bQARowStopperMotorFwd1:=FALSE;
bQARowStopperMotorFwd2:=FALSE;
bQARowStopperMotorFwd3:=FALSE;
bQARowStopperMotorRev1:=FALSE;
bQARowStopperMotorRev2:=FALSE;
bQARowStopperMotorRev3:=FALSE;
bQARowStopperMotorRevAuto:=FALSE;
bRowStopperGoRst:=FALSE;
step2:=0;
step1:=0;
step3:=0;
step4:=0;

END_IF
END_PROGRAM

(* POU Auto/ColumStopperMotor, ST *)
PROGRAM ColumStopperMotor
VAR
	bQAColumnStopperMotorFwd1: BOOL;
	bQAColumnStopperMotorRev1: BOOL;
	step1: INT;

	test: BOOL;

	step2: INT;
	ColumnStopperInHome: BOOL;
	bA4_4MoveStarted: BOOL;
	bQAColumnStopperMotorFw21: BOOL;
	bQAColumnStopperMotorFwd2: BOOL;
	bQAColumnStopperMotorRev2: BOOL;
	bQAColumnStopperMotorFw2: BOOL;
	test1: BOOL;
	step3: INT;
	test2: BOOL;
	bA2_3MoveStarted: BOOL;
	bQAColumnStopperMotorRev3: BOOL;
	bQAColumnStopperMotorFwd3: BOOL;
	RevOffDly: TON;
	bA2_4MoveStarted: BOOL;
	Timer1: TON;
	Timer2: TON;
	bStopHmitemp: BOOL;
	bProgramChange: BOOL;
	bColumnStopMove2_3: BOOL;
	bColumnStopMove2_4: BOOL;
	b2_3SetHmiSelectedtemp: BOOL;
	b2_4SetHmiSelectedtemp: BOOL;
	b2_4SetHmiSelectedtemp1: BOOL;
	Mybit1: BOOL;
END_VAR
bQAColumnStopperMotorForward:= ( bQAColumnStopperMotorFwd1 OR bQAColumnStopperMotorFwd2 OR bQAColumnStopperMotorFwd3  ) ;
bQAColumnStopperMotorReverse:= ( bQAColumnStopperMotorRev1 ) ;

								(*=========== Column Stopper Motor Home Position Logic===============*)

CASE step2 OF

	0:	IF  bInitializeHmi AND NOT bIColumnStopperHome  AND NOT bAinterlockinit   THEN
		bQAColumnStopperMotorFwd1:=TRUE;
		(*	Timer1(IN:=TRUE  , PT:=t#1s , Q=> , ET=> );   *) step2:=step2+1;
		ELSIF  bInitializeHmi AND  bIColumnStopperHome    THEN   step2:=4;
		END_IF

	1:	bQAColumnStopperMotorFwd1:=FALSE;
		Timer2(IN:=TRUE , PT:= t#0.5s, Q=> , ET=> );
		IF Timer2.Q THEN step2 :=step2+1; END_IF

	2:	IF NOT bAPauseSeq  THEN  bQAColumnStopperMotorRev1:=TRUE; step2:=step2+1; END_IF

	3:	IF bIColumnStopperHome THEN bQAColumnStopperMotorRev1:=FALSE; step2:=step2+1; END_IF

	4:	IF b2_3SetHmiSelected THEN bColumnStopMove2_3:=TRUE; step2:=0;
		ELSIF b2_4SetHmiSelected THEN bColumnStopMove2_4:=TRUE; step2:=0;
		END_IF

END_CASE

										(*=========== Column Stopper Motor 2_3 Position Logic===============*)

CASE step1 OF

	0:	IF  b2_3SetHmiSelected AND bColumnStopMove2_3 AND NOT bIColumnStopper3  AND  bIColumnStopperHome  THEN
		 bQAColumnStopperMotorFwd2:=TRUE; step1:=step1+1;
		END_IF

	1:	IF bIColumnStopper3 THEN
	         bColumnStopMove2_3:=FALSE;
                  bQAColumnStopperMotorFwd2:=FALSE; step1:=step1+1;
		END_IF

	2:	 step1:=0;

END_CASE

										(*=========== Column Stopper Motor 2_4 Position Logic===============*)

CASE step3 OF

	0:	IF b2_4SetHmiSelected AND  bColumnStopMove2_4 AND NOT bIColumnStopper2  AND    bIColumnStopperHome   THEN
		bQAColumnStopperMotorFwd3:=TRUE; step3:=step3+1;
		END_IF


	1: 	IF bIColumnStopper2 THEN
		bColumnStopMove2_4:=FALSE;
		bQAColumnStopperMotorFwd3:=FALSE; step3:=step3+1;
		END_IF


	2:	step3:=0;

END_CASE
END_PROGRAM

(* POU StartUp/GripperUnitRst, ST *)
PROGRAM GripperUnitRst
VAR
	step: INT;
	bILengthTightPistonEnd: BOOL;
	bIBredthTightPistonEnd: BOOL;
	bEmptyCortonConveyoPiatonHome: BOOL;
	bHorPistonAtReadyPos: BOOL;
	bHorPistonAtHomePos: BOOL;
	bHorPistonAtMiddlePos: BOOL;
	bGripperAtHomePos: BOOL;
	bGripperAtEndPos: BOOL;
	bGripperAtMiddlePos: BOOL;
	bSepVerticalAtHomePos: BOOL;
	bSepVerticalAtEndPos: BOOL;
	bSepVerticalAtMiddlePos: BOOL;
	bLenghtTightPistonHomeNok: BOOL;
	bBreathtightPistonHomeNok: BOOL;
	bApplicatorHomeNok: BOOL;
	bReleaseApplicator: BOOL;
	step2: INT;
	Timer1: TON;
	Timer2: TON;
	Timer3: TON;
	Timer4: TON;
	ReadyToRelease: BOOL;
	Timer5: TON;
	bAResetHmitemp: BOOL;
	Timer6: TON;
	Timer7: TON;
	Timer8: TON;
	Timer9: TON;
	test: BOOL;
END_VAR
VAR_INPUT
END_VAR
IF bInitializeHmi AND bAutoModeOn AND bMCStartInAuto THEN
step:=0;
END_IF



CASE step OF
	0:	iControlWord1.7:=TRUE;
		 bHomingDone:=FALSE;
		step:=step+1;

	1:	 iControlWord1.7:=FALSE;
		step:=step+1;


	2:	IF  bAResetHmitemp OR bMatrixConvIntOver THEN step:=step+1;  END_IF

	3:	IF NOT bIGripperVerticalHome THEN   bRServoHome:=TRUE; step:=step+1;
		ELSIF bIGripperVerticalHome  THEN step:=5;
		END_IF

	4:	IF bHomingDone THEN step:=step+1; END_IF

	5:	bMatrixConvIntOver:=FALSE;
		bHomingDone:=FALSE; (*bRowStopperGoHome:=TRUE;*)
		step:=step+1;

	6:	IF bISeparatorHorizontalPistonEnd AND NOT  bISeparatorHorizontalPistonHome THEN
		bHorPistonAtReadyPos:=TRUE; bHorPistonAtHomePos:=FALSE; bHorPistonAtMiddlePos:=FALSE;
		step:=step+1;
		ELSIF NOT bISeparatorHorizontalPistonEnd  AND  bISeparatorHorizontalPistonHome THEN
		bHorPistonAtHomePos:=TRUE; bHorPistonAtReadyPos:=FALSE; bHorPistonAtMiddlePos:=FALSE;
		step:=step+1;
		ELSIF NOT bISeparatorHorizontalPistonEnd  AND  NOT bISeparatorHorizontalPistonHome THEN
		bHorPistonAtMiddlePos:=TRUE; bHorPistonAtHomePos:=FALSE; bHorPistonAtReadyPos:=FALSE;
		step:=step+1;
		END_IF

	7:	IF bHorPistonAtReadyPos THEN step:=8;
		ELSIF bHorPistonAtHomePos THEN step:=25;
		ELSIF bHorPistonAtMiddlePos THEN  step:=25; END_IF

	8:	 iControlWord1:=0;
		step:=step+1;

	9:	 iControlWord1:=6;
		step:=Step+1;
(*========Waiting for row stopper to home==========*)

	10:	IF bIRowStopperHome THEN step:=Step+1;
		ELSIF NOT bIRowStopperHome THEN bRowStopperGoHome:=TRUE;  step:=Step+1;  END_IF


	11:	IF  bIRowStopperHome THEN iControlWord1:=7;
		bHomingDone:=FALSE;
		step:=Step+1;
		END_IF

	12:	IF ModeACT=1THEN  step:=15;
		ELSIF  ModeACT<>1 THEN step:=Step+1;
		END_IF

	13:	ModeWrite:=1;
		step:=Step+1;

	14:	bAModeWrite:=TRUE;
		Timer1(IN:=TRUE , PT:=T#100ms , Q=> , ET=> );
		IF Timer1.Q THEN step:=Step+1;  END_IF


	15:	diTargetVelocity1:=rPickVeloFinal;
		diTargetPosition:=-87947 ; (*rTargetPosFinal*);
		bAModeWrite:=FALSE;
		step:=Step+1;

	16:	Timer2(IN:=TRUE , PT:= t#100ms, Q=> , ET=> );
		IF Timer2.Q THEN  step:=Step+1; END_IF

	17:	iControlWord1:=15;
		step:=Step+1;

	18:	Timer3(IN:=TRUE , PT:= t#1s, Q=> , ET=> );
		IF Timer3.Q  THEN step:=Step+1; END_IF

	19:	IF statusWord.2 THEN    iControlWord1.4:=TRUE;
		step:=Step+1;
		END_IF
	20:	Timer4(IN:=TRUE , PT:= t#5s, Q=> , ET=> );
		IF Timer4.Q THEN iControlWord1.4:=FALSE; step:=Step+1; END_IF

	21:	IF statusWord.10 THEN step:=Step+1; END_IF

	22:	bQABreadthTightPistonValve:=FALSE;
		bQALengthTightPistonValve:=FALSE;
		bQMBreadthTightPistonValve:=FALSE;
		bQMLengthTightPistonValve:=FALSE;
		 step:=Step+1;

	23:	IF(* bILengthTightPistonHome AND*) bIBreadthTightPistonHome AND bIGripperVerticalEnd   THEN  step:=Step+1; END_IF

	24:	bRServoHome:=TRUE;
		IF bHomingDone THEN bGripperUnitOver:=TRUE;  step:=0; END_IF

(*========Reseting all auto and manual output and enabling Rst outpus===================*)

	25:	IF bIGripperVerticalHome THEN bQASeparatorHorizontalPistonValveFWD:=FALSE;
		bQASeparatorHorizontalPistonValveREV:=FALSE;
		bQMSeparatorHorizontalPistonValveRev:=FALSE;
		bQMSeparatorHorizontalPistonValveFwd:=FALSE;
		bHomingDone:=FALSE;
		step:=step+1;
		END_IF

	26:	bQRSeparatorHorizontalPistonValveREV:=TRUE;
		step:=step+1;

	27:	IF bISeparatorHorizontalPistonEnd THEN bReleaseApplicator:=TRUE; bQRSeparatorHorizontalPistonValveREV:=FALSE; step:=step+1; END_IF


	28:	IF ReadyToRelease THEN	step:=step+1; 	END_IF

	29:	Timer5(IN:=TRUE , PT:=t#1s , Q=> , ET=> );
		IF Timer5.Q THEN ReadyToRelease:=FALSE; step:=step+1; 	END_IF

	30:	bQMBreadthTightPistonValve:=FALSE;
		bQMLengthTightPistonValve:=FALSE;
		bQABreadthTightPistonValve:=FALSE;
		bQALengthTightPistonValve:=FALSE;
		step:=step+1;

	31:	IF bIBreadthTightPistonHome(* AND bILengthTightPistonHome*) THEN
		bRServoHome1:=TRUE;
		IF bHomingDone THEN bGripperUnitOver:=TRUE;  step:=0; END_IF
		END_IF


END_CASE




CASE step2 OF

	0:	IF bReleaseApplicator  THEN
		Timer6(IN:=FALSE);
		Timer7(IN:=FALSE);
		step2:=step2+1;
		END_IF

	1:	IF bIRowStopperHome THEN step2:=step2+1;
		ELSIF NOT bIRowStopperHome THEN  bRowStopperGoHome1:=TRUE;  step:=Step+1;  END_IF


	2: 	IF bIRowStopperHome  THEN   iControlWord1:=7;
		bReleaseApplicator:=FALSE;
		Timer8(IN:=FALSE);
		step2:=step2+1;
		END_IF

	3:	Timer6(IN:=TRUE , PT:=T#100ms , Q=> , ET=> );
		IF Timer6.Q THEN
		step2:=step2+1;
		END_IF

	4:	IF NOT bIGripperVerticalEnd AND bIRowStopperHome THEN
		ModeWrite:=3;							(*=========Changing the servo Mode to Velocity mode=============*)
		Timer8(IN:=FALSE);
		Timer9(IN:=FALSE);

		step2:=step2+1;
		END_IF

	5:	Timer7(IN:=TRUE , PT:=T#100ms , Q=> , ET=> );
		IF Timer7.Q THEN
		step2:=step2+1;
		END_IF


	6:	bAModeWrite:=TRUE;
		Timer8(IN:=TRUE , PT:=T#100ms , Q=> , ET=> );
		IF Timer8.Q THEN
		step2:=step2+1;
		END_IF

	7:	IF ModeWrite = ModeAct THEN
		bAModeWrite:=FALSE;
		step2:=step2+1;
		END_IF

	8:	IF  statusWord.1 THEN iControlWord1 :=15;
		Timer9(IN:=TRUE , PT:=T#1s , Q=> , ET=> );
		IF Timer9.Q THEN
		step2:=step2+1;
		END_IF
		END_IF

	9:	diTargetVelocity:=-100;
		step2:=step2+1;


	10:	IF statusWord.2 THEN
		iControlWord1.4:= TRUE;
		step2:=step2+1;
		END_IF




	11:	IF bIGripperVerticalEnd THEN
		iControlWord1.4 := FALSE;
		iControlWord1:=7;
		diTargetVelocity:=0;
		step2:=step2+1;
		END_IF

	12: 	Timer6(IN:=FALSE);
		Timer7(IN:=FALSE);
		Timer8(IN:=FALSE);
		Timer9(IN:=FALSE);
		step2:=step2+1;

	13:	ReadyToRelease:=TRUE;
		step2:=0;




END_CASE


IF NOT bIEmergencySwitch OR bStopHmi OR bIMcStop OR bServoOff  THEN

bRServoHome:=FALSE;
bHorPistonAtReadyPos:=FALSE;
bHorPistonAtHomePos:=FALSE;
bHorPistonAtMiddlePos:=FALSE;
bAModeWrite:=FALSE;
Timer1(IN:=FALSE);
Timer2(IN:=FALSE);
Timer3(IN:=FALSE);
Timer4(IN:=FALSE);
bRServoHome:=FALSE;
bQRSeparatorHorizontalPistonValveREV:=FALSE;
Timer5(IN:=FALSE);
bRServoHome1:=FALSE;
bReleaseApplicator:=FALSE;
bGripperUnitOver:=FALSE;
Timer6(IN:=FALSE);
Timer7(IN:=FALSE);
Timer8(IN:=FALSE);
Timer9(IN:=FALSE);
iControlWord1.4:= FALSE;
ReadyToRelease:=FALSE;
iControlWord1:=7;
step:=0;
step2:=0;

END_IF
END_PROGRAM

(* POU Serial, ST *)
PROGRAM Serial
VAR
	bSendStr:BOOL;
	Timer: TON;
	TrigSend:R_TRIG;
	TransmitStr : SendString;
	SendBusy: BOOL;
	SendErrorID: ComError_t;

	ReceiveStr :ReceiveString;
	ReStr: STRING;
	LastReceivedString: STRING;
	StringReceived: BOOL;
	ReceiveBusy: BOOL;
	ReceiveError: BOOL;
	ReceiveErrorID: ComError_t;
	ReceiveTimeout: BOOL;
	ReceiveCounter: UDINT;

	(* Serial communication with the COM port device *)
	COMportControl: SerialLineControl;
	COMportControlError: BOOL;
	COMportControlErrorID: ComError_t;


	Decimaldata: BYTE;
	Stringdata: STRING;
	RxBufferStringdata: STRING(300);
	TxBufferStringdata: STRING(300);
	RxBufferArrdata: ARRAY [0..80] OF BYTE;
	TxBufferArrdata: ARRAY [0..80] OF BYTE :=(*16#0F, 16#FA, 16#03, 16#00, 16#0D, 16#00, 16#10, 16#20, 16#01, 16#05, 16#58, 16#DF, 16#98, 16#00, 16#00, 16#02, 16#04, 16#E0, 16#B4, 16#F0;*)
16#0F, 16#FA, 16#03, 16#00, 16#02, 16#00, 16#38, 16#24, 16#F0; (*16#00, 16#00, 16#00, 16#00;, 16#10, 16#20, 16#05, 16#02, 16#AF, 16#F6, 16#98, 16#00, 16#00, 16#02, 16#04, 16#E0, 16#84, 16#F0;*)
	i: INT;
	ReceiveData_1: ReceiveData;

	SReceivedataFormat: ARRAY [0..300] OF BYTE;
	SReceivedatStringFt: STRING(300);
	sSendString_1: STRING(300);
	TransmitArrByteData: SendData;
(*==============port 2==========*)
	ReceiveData_2: ReceiveData;

	test: BOOL;
	SReceivedataFormat_2: ARRAY [0..300] OF BYTE;
	SReceivedatStringFt_2: STRING(300);
	COMportControl_2: SerialLineControl;
	COMportControlError_2: BOOL;
	COMportControlErrorID_2: ComError_t;
	SReceivedatStringFtTemp: STRING;
	SReceivedatStringFt_2Temp: STRING(80);
	ReceiveData_3: ReceiveData;
	SReceivedataFormat_3: ARRAY [0..300] OF BYTE;
	SReceivedatStringFt_3: STRING(300);
	SReceivedatStringFt_3Temp: STRING;
	COMportControl_3: SerialLineControl;
	COMportControlError_3: BOOL;
	COMportControlErrorID_3: ComError_t;

	prefix_data: BYTE ;
	sufix_data: BYTE;
	samplestring: STRING;
	ReceiveString_sample: ReceiveString;
	ipos: INT;
	resultWt: STRING;
END_VAR
(*
TrigSend(CLK:=bSendStr , Q=> );

Timer(IN:=TRUE, PT:=T#1s);


IF TrigSend.Q THEN
	TransmitArrByteData(
	pSendData:= ADR(TxBufferArrdata),
	Length:=100 ,
	TXbuffer:= TxBuffer1,
	Busy=> ,
	Error=> );

	Timer(IN:=FALSE);

END_IF;



MEMCPY(ADR(sSendString), ADR(TxBufferArrdata), 50);
*)
(*==============El6002 serial Communication Program for Laod Cell value read in Rs232 port 1 ==================*)


COMportControl(
	Mode:= SERIALLINEMODE_EL6_22B,
	pComIn:= ADR(COMin_COMport),
	pComOut:= ADR(COMout_COMport),
	SizeComIn:= SIZEOF(COMin_COMport),
	TxBuffer:= TxBuffer1,
	RxBuffer:= RxBuffer1,
	Error=> COMportControlError,
	ErrorID=> COMportControlErrorID );



ReceiveString_sample(
	Prefix:='w' ,
	Suffix:='g' ,
	Timeout:= t#5s,
	Reset:= ,
	ReceivedString:=samplestring ,
	RXbuffer:= RxBuffer1,
	StringReceived=> ,
	Busy=> ,
	Error=> ,
	RxTimeout=> );
ipos:=FIND(samplestring,'n');

resultWt:= MID (samplestring,9,ipos+1);

rRetUnitAWeight:=STRING_TO_REAL(resultWt);

(************************************
MAIN.string_Dec();

***)



(*
FOR i:=0 TO 300 DO
	RxBufferStringData[i]:= RxBuffer1.Buffer[i];
END_FOR*)
(********************************test
ReceiveData_1(
	pPrefix:= ,
	LenPrefix:= ,
	pSuffix:= ,
	LenSuffix:= ,
	pReceiveData:=  ADR(SReceivedataFormat),
	SizeReceiveData:= 100,
	Timeout:=t#1s ,
	Reset:= ,
	RXbuffer:=RxBuffer1 ,
	DataReceived=> ,
	busy=> ,
	Error=> ,
	RxTimeout=> ,
	LenReceiveData=> );*********************************)
(*************************************
ReceiveString_sample(
	Prefix:='w' ,
	Suffix:='g' ,
	Timeout:= t#5s,
	Reset:= ,
	ReceivedString:=samplestring ,
	RXbuffer:= RxBuffer2,
	StringReceived=> ,
	Busy=> ,
	Error=> ,
	RxTimeout=> );
ipos:=FIND(samplestring,'n');*)
(****************************************test************
MEMCPY(ADR(SReceivedatStringFt), ADR(SReceivedataFormat), 50);

SReceivedatStringFtTemp:=MID(STR:=SReceivedatStringFt, LEN:=7, POS:=3);


 rRetUnitAWeight:=STRING_TO_REAL (SReceivedatStringFtTemp);**********************************************test*)

(*==============El6002 serial Communication Program for Laod Cell value read in Rs232 port 2 ==================*)

COMportControl_2(
	Mode:= SERIALLINEMODE_EL6_22B,
	pComIn:= ADR(COMin_2_COMport_2),
	pComOut:= ADR(COMout_2_COMport_2),
	SizeComIn:= SIZEOF(COMin_2_COMport_2),
	TxBuffer:= TxBuffer2,
	RxBuffer:= RxBuffer2,
	Error=> COMportControlError_2,
	ErrorID=> COMportControlErrorID_2 );






ReceiveData_2(
	pPrefix:= ,
	LenPrefix:= ,
	pSuffix:= ,
	LenSuffix:= ,
	pReceiveData:=  ADR(SReceivedataFormat_2),
	SizeReceiveData:= 100,
	Timeout:=t#1s ,
	Reset:= ,
	RXbuffer:=RxBuffer2 ,
	DataReceived=> ,
	busy=> ,
	Error=> ,
	RxTimeout=> ,
	LenReceiveData=> );

MEMCPY(ADR(SReceivedatStringFt_2), ADR(SReceivedataFormat_2), 50);

 rRetUnitBWeight:=STRING_TO_REAL (SReceivedatStringFt_2);


SReceivedatStringFt_2Temp:=MID(STR:=SReceivedatStringFt_2, LEN:=7, POS:=3);


 rRetUnitBWeight:=STRING_TO_REAL (SReceivedatStringFt_2Temp);



(*==============El6002 serial Communication Program for Laod Cell value read in Rs232 port 2 (  GROSS WEIGHT    )  ==================*)

COMportControl_3(
	Mode:= SERIALLINEMODE_EL6_22B,
	pComIn:= ADR(COMin_3_COMport_3),
	pComOut:= ADR(COMout_3_COMport_3),
	SizeComIn:= SIZEOF(COMin_3_COMport_3),
	TxBuffer:= TxBuffer3,
	RxBuffer:= RxBuffer3,
	Error=> COMportControlError_3,
	ErrorID=> COMportControlErrorID_3 );





ReceiveData_3(
	pPrefix:= ,
	LenPrefix:= ,
	pSuffix:= ,
	LenSuffix:= ,
	pReceiveData:=  ADR(SReceivedataFormat_3),
	SizeReceiveData:= 100,
	Timeout:=t#1s ,
	Reset:= ,
	RXbuffer:=RxBuffer3 ,
	DataReceived=> ,
	busy=> ,
	Error=> ,
	RxTimeout=> ,
	LenReceiveData=> );

MEMCPY(ADR(SReceivedatStringFt_3), ADR(SReceivedataFormat_3), 50);




SReceivedatStringFt_3Temp:=MID(STR:=SReceivedatStringFt_3, LEN:=7, POS:=3);


 rGrossWeight:=STRING_TO_REAL (SReceivedatStringFt_3Temp);
END_PROGRAM

(* POU Auto/Gripper/Servo_Auto, ST *)
PROGRAM Servo_Auto
VAR
	step: INT;




	bAServoDownDone1: BOOL;

	iAServoRevVelocityHmi: UINT := 6000;
	bAServoFwdStart1: BOOL;
	test: BOOL;


	step2: INT;
	test2: BOOL;
	test3: BOOL;



	iTargetCounter: UDINT;
	TON_1: TON;
	TON_2: TON;
	TON_3: TON;
	TON_4: TON;
	TON_5: TON;
	TON_6: TON;
	TON_7: TON;
	bIGripperVerticalHomeTemp: BOOL;
	bIBreadthTightPistonHomeTemp: BOOL;
	bILengthTightPistonHomeTemp: BOOL;
	bAServoFwdStartTemp: BOOL;
	EnableTemp: BOOL;
	bAServoFwdStartTemp2: BOOL;
	bIGripperVerticalHomeTemp2: BOOL;
	bILengthTightPistonHomeTemp2: BOOL;
	bIBreadthTightPistonHomeTemp2: BOOL;
	diTargetPositionHmi: DINT;
	diTargetVelocityHmi: DINT := 200;
	TON_8: TON;
	TON_9: TON;
	TON_10: TON;
	TON_11: TON;
	TON_12: TON;
	TON_13: TON;
	TON_14: TON;
	TON_15: TON;
	TON_16: TON;
	TON_17: TON;
	TON_18: TON;
	TON_19: TON;
	TON_20: TON;
	TON_21: TON;
	TON_22: TON;
	TON_23: TON;
	TON_24: TON;
	TON_25: TON;
	TON_26: TON;
	TON_27: TON;
	TON_28: TON;
	bServoPauseActive1: BOOL;
	bServoReumeActive1: BOOL;
	bAServoFwdStartAuto: BOOL;
	R_TRIG_1: R_TRIG;
	bServoFirstStart: BOOL;
	bPauseOperationEn1: BOOL;
	bPauseOperationEn2: BOOL;
	bPauseOperationEn3: BOOL;
	bServoPauseActive2: BOOL;
	bServoReumeActive2: BOOL;
	R_TRIG_2: R_TRIG;
	bServoPauseActive3: BOOL;
	bServoReumeActive3: BOOL;
	R_TRIG_3: R_TRIG;

	bPauseOperationEn5: BOOL;
	bServoPauseActive5: BOOL;
	bServoReumeActive5: BOOL;
	R_TRIG_: BOOL;
	R_TRIG_5: R_TRIG;
	TON_29: TON;
	TON_30: TON;
	bPauseOperationEn6: BOOL;
	bServoPauseActive6: BOOL;
	bServoReumeActive6: BOOL;
	R_TRIG_6: R_TRIG;
	CTU_test: CTU;
	temp11: BOOL;
	temp15: BOOL;
	temp19: BOOL;
	temp20: BOOL;


END_VAR
IF bISeparatorHorizontalPistonEnd AND bIRowStopperHome AND bAutoModeOn AND bIGripperConeDetection THEN
bAGripperConeAllignError:=TRUE;bAGripCheckDownBuzzer:=TRUE;sMessage_ServoGripperDown:='  Check Cone Allign at Gripper Bottom ';END_IF
IF bErrorReset AND NOT bIGripperConeDetection THEN sMessage_ServoGripperDown:='   ';bAGripperConeAllignError:=FALSE;bAGripCheckDownBuzzer:=FALSE;END_IF

CASE step OF

	0:	IF bAServoFwdStart  AND bAutoModeOn  AND bIGripperVerticalHome AND bISeparatorHorizontalPistonEnd AND NOT bAGripperConeAllignError
		AND (* bILengthTightPistonHome AND*) bIBreadthTightPistonHome AND bIRowStopperHome AND NOT  bIRowStopper2
		AND NOT  bIRowStopper3   THEN
		bHomingDone:=FALSE;

		TON_7(IN:=FALSE);
		TON_1(IN:=FALSE);
		TON_15(IN:=FALSE);

		step:=Step+1;
		END_IF     sMessage_Gripper:='  Check Lenght & Breadth & Vertical & Row Stopper Home ';

	1:	IF ModeACT=1THEN step:=4;
		ELSIF  ModeACT<>1 THEN step:=Step+1;
		END_IF

	2:	iControlWord1:=7;
		ModeWrite:=1;
		bAServoFwdStart:=FALSE;
		step:=Step+1;

	3:	bAModeWrite:=TRUE;
		bServoPauseActive1:=FALSE;
		bServoReumeActive1:=FALSE;
		TON_7(IN:=TRUE , PT:=T#100ms , Q=> , ET=> );
		IF TON_7.Q THEN step:=Step+1;  END_IF


	4:	diTargetVelocity1:=rPickVeloFinal;(*need to add velo var*)
		diTargetPosition:=  -87947 ; (*rTargetPosFinal;*)
		bAModeWrite:=FALSE;
		TON_2(IN:=FALSE);
		step:=Step+1;

	5:	TON_1(IN:=TRUE , PT:= t#100ms, Q=> , ET=> );
		IF TON_1.Q THEN  step:=Step+1; END_IF

	6:	iControlWord1:=15;
		bAServoFwdStart:=FALSE;
		TON_3(IN:=FALSE);
		step:=Step+1;

	7:	IF statusWord.2 THEN TON_2(IN:=TRUE , PT:= t#0.1s, Q=> , ET=> );
		IF TON_2.Q   AND NOT bAPauseSeq    THEN step:=Step+1; END_IF  END_IF

	8:	iControlWord1.4:=TRUE;
		TON_22(IN:=FALSE) ;
		TON_18(IN:=FALSE) ;
		TON_19(IN:=FALSE) ;
		TON_20(IN:=FALSE) ;
		TON_21(IN:=FALSE) ;
		step:=Step+1;


	9:	TON_3(IN:=TRUE , PT:= t#2s, Q=> , ET=> );  (* === old time value  PT:= t#5s====*)
		IF TON_3.Q THEN iControlWord1.4:=FALSE;bChkEndSensor:=TRUE;  step:=  24; END_IF   (* old Step no step:=  step+1;*)
(*====newly added for checking  from step 10 to step 15=========*)

	10:	IF statusWord.10 AND rServiActPosHmi <= -540 THEN   iControlWord1:=0; step:=Step+1; END_IF

	11:	IF  NOT  statusWord.12 THEN
		diTargetPosition:=-71022 ;                  (*==============  Pulse for 740 mm =========  -86947======*)
		diTargetVelocity1:=100;
		TON_22(IN:=TRUE , PT:= t#100ms , Q=> , ET=> );
		IF TON_22.Q THEN step:=Step+1; END_IF
		 step:=Step+1;
		END_IF


	12:	 iControlWord1:=6;
		TON_18(IN:=TRUE , PT:= t#100ms , Q=> , ET=> );
		IF TON_18.Q THEN step:=Step+1; END_IF


	13:	 iControlWord1:=7;
		TON_19(IN:=TRUE , PT:= t#50ms , Q=> , ET=> );
		IF TON_19.Q THEN step:=Step+1; END_IF


	14:	 IF statusWord.1 THEN  iControlWord1:=15;
		bServoPauseActive2:=FALSE;
		bServoReumeActive2:=FALSE;
		TON_20(IN:=TRUE , PT:= t#100ms , Q=> , ET=> );
		IF TON_20.Q THEN bServoStartedInAuto:=TRUE; step:=Step+1; END_IF END_IF



	15:	IF statusWord.2 THEN  iControlWord1.4:=TRUE;

		TON_21(IN:=TRUE , PT:= t#3s, Q=> , ET=> );
		IF TON_21.Q THEN step:=Step+1; END_IF
		END_IF


(*====================  logic for third high speed================*)

	16:	IF statusWord.10 AND  rServiActPosHmi <= -596 THEN   iControlWord1:=0; step:=Step+1; END_IF

	17:	TON_23(IN:=FALSE) ;
		TON_24(IN:=FALSE) ;
		TON_25(IN:=FALSE) ;
		TON_26(IN:=FALSE) ;
		TON_27(IN:=FALSE) ;
		step:=Step+1;


	18:	 iControlWord1.4:=FALSE;
		step:=Step+1;



	19:	IF  NOT  statusWord.12 THEN
		diTargetPosition:=-87947 ;                  (*==============  Pulse for 740 mm =========  -86947======*)
		diTargetVelocity1:=rPickVeloFinal;
		TON_23(IN:=TRUE , PT:= t#100ms , Q=> , ET=> );
		IF TON_23.Q THEN step:=Step+1; END_IF
		 step:=Step+1;
		END_IF


	20:	 iControlWord1:=6;
		bServoStartedInAuto:=FALSE;
		TON_24(IN:=TRUE , PT:= t#100ms , Q=> , ET=> );
		IF TON_24.Q THEN step:=Step+1; END_IF


	21:	 iControlWord1:=7;
		TON_25(IN:=TRUE , PT:= t#100ms , Q=> , ET=> );
		IF TON_25.Q THEN step:=Step+1; END_IF


	22:	 iControlWord1:=15;
		bServoReumeActive3:=FALSE;
		bServoReumeActive3:=FALSE;
		TON_26(IN:=TRUE , PT:= t#100ms , Q=> , ET=> );
		IF TON_26.Q THEN step:=Step+1; END_IF



	23:	IF statusWord.2 THEN  iControlWord1.4:=TRUE;
		TON_27(IN:=TRUE , PT:= t#1s, Q=> , ET=> );  (* old time Val === PT:= t#2s*)
		IF TON_27.Q THEN step:=Step+1; END_IF
		END_IF




	24:	IF statusWord.10 THEN       (*==========old step no was 10===========*)
		 iControlWord1.4:=FALSE;
		TON_16(IN:=FALSE);
		TON_4(IN:=FALSE);
		TON_17(IN:=FALSE);
		step:=Step+1;
		END_IF


	25:	IF bIGripperVerticalEnd  THEN
		TON_15(IN:=TRUE , PT:=t#0.1s , Q=> , ET=> );  (*old time Val PT:=t#1s*)
		sMessage_Gripper:='  Check Gripper Vertical End Reed Switch ';
		IF	TON_15.Q THEN bChkEndSensor:=FALSE;  Step:=Step+1; END_IF                    	(*	iControlWord1:=6;    *)
		END_IF

	26:     iControlWord1:=0;
		bAServoDownDone:=TRUE;
		bServoStartedInAuto:=FALSE;
		TON_16(IN:=TRUE , PT:=t#50ms , Q=> , ET=> );
		IF TON_16.Q THEN  step:=Step+1; END_IF

	27:	IF bAConePickDone  THEN

		TON_5(IN:=FALSE);
		TON_6(IN:=FALSE);
		TON_16(IN:=FALSE);
		step:=Step+1;
		END_IF




	28:	 iControlWord1:=6;
		TON_17(IN:=TRUE , PT:= T#0.1s, Q=> , ET=> );  (*=== PT:= T#1s  ===*)
		IF TON_17.Q THEN step:=Step+1; END_IF


	29:	  iControlWord1:=7;
		 IF statusWord.1 THEN step:=Step+1; END_IF   (*    newly added for time reduce=====*)



	30:	IF NOT  statusWord.12 THEN
		 iControlWord1:=15;
		TON_4(IN:=TRUE , PT:= T#100ms, Q=> , ET=> );  (* bASrevoAutoHome:=TRUE; *)
		IF TON_4.Q THEN TON_5(IN:=FALSE);  TON_6(IN:=FALSE);  Step:=Step+1; END_IF
		END_IF

	31:	diTargetVelocity1:=2000;
		diTargetPosition:=0;
		TON_6(IN:=FALSE);
		bAConePickDone:=FALSE;
		TON_17(IN:=FALSE);
		step:=Step+1;


	32:	Step:=Step+1;


	33:	 IF statusWord.2 THEN
		TON_5(IN:=TRUE , PT:= T#50ms, Q=> , ET=> );
		IF TON_5.Q   THEN Step:=Step+1; END_IF
		END_IF


	34:	iControlWord1.4:=TRUE;
		step:=Step+1;

	35:	step:=Step+1;

	36:
		TON_6(IN:=TRUE , PT:= t#4s, Q=> , ET=> );
		IF TON_6.Q THEN step:=Step+1; END_IF




	37:	IF statusWord.10  AND bIGripperVerticalHome   THEN
		 iControlWord1.4:=FALSE;
		bServoReachedUp:=TRUE;
		step:=Step+1;
		END_IF  sMessage_Gripper:='  Check Vertical  Home Reed Switch ';

	38:	iControlWord1:=7;

		step:=Step+1;

	39:	TON_1(IN:=FALSE);
		TON_2(IN:=FALSE);
		TON_3(IN:=FALSE);
		TON_4(IN:=FALSE);
		TON_5(IN:=FALSE);
		TON_6(IN:=FALSE);
		TON_7(IN:=FALSE);
		TON_15(IN:=FALSE);
		step:=0;


END_CASE









CASE step2 OF

	0:	IF bAServoFwdStart2 AND bAutoModeOn  AND bIGripperVerticalHome AND NOT bHmiColourChangeBit2_24
		AND (*NOT  bILengthTightPistonHome AND *)NOT bIBreadthTightPistonHome  THEN
		bHomingDone:=FALSE;
		TON_8(IN:=FALSE);
		TON_9(IN:=FALSE);
		iControlWord1:=7;
		step2:=Step2+1;
		END_IF  sMessage_Gripper:='  Check Lenght & Breadth & Vertical & Row Stopper Home ';

	1:	IF ModeACT=1THEN step2:=4;
		ELSIF  ModeACT<>1 THEN step2:=Step2+1;
		END_IF

	2:	ModeWrite:=1;
		step2:=Step2+1;

	3:	bAModeWrite:=TRUE;
		TON_8(IN:=TRUE , PT:=T#500ms , Q=> , ET=> );
		IF TON_8.Q THEN step2:=Step2+1;  END_IF

	4: 	 diTargetVelocity1:=REAL_TO_DINT (rDropVeloFinal);
		diTargetPosition:=REAL_TO_DINT ( rDropPosFinal ) ;
		bAModeWrite:=FALSE;
		TON_9(IN:=FALSE);
		step2:=Step2+1;

	5:	TON_9(IN:=TRUE , PT:= t#100ms, Q=> , ET=> );
		IF TON_9.Q   THEN  step2:=Step2+1; END_IF

	6:	iControlWord1:=15;
		TON_11(IN:=FALSE);
		step2:=Step2+1;

	7:	TON_10(IN:=TRUE , PT:= t#1s, Q=> , ET=> );
		IF TON_10.Q AND statusWord.2 THEN step2:=Step2+1; END_IF

	8:	 IF NOT  bAPauseSeq THEN    iControlWord1.4:=TRUE; temp11:=TRUE;
		TON_11(IN:=TRUE , PT:= t#3s, Q=> , ET=> );bAServoFwdStart2:=FALSE;
		IF TON_11.Q THEN  step2:=Step2+1; END_IF END_IF

	9:	IF statusWord.10 THEN
		iControlWord1.4:=FALSE;
		TON_12(IN:=FALSE);
		 temp11:=FALSE;
		step2:=Step2+1;
		END_IF

	10:	(*IF bIGripperVerticalEndtemp THEN  *)
		step2:=Step2+1;


	11:	 iControlWord1:=0;                                   (*-========== iControlWord1:=6;  old value=============*)
		bAServoDown1Done:=TRUE;
		step2:=Step2+1;

	12:	step2:=Step2+1;


	13:	TON_12(IN:=TRUE , PT:= T#1s, Q=> , ET=> );  (* bASrevoAutoHome:=TRUE; *)  (*  Old Value=====PT:= T#2s   *)
		IF TON_12.Q THEN Step2:=Step2+1; END_IF


	14:	IF bAServoUpAuto THEN
		diTargetVelocity1:=2500;
		diTargetPosition:=0;
		step2:=Step2+1;
		END_IF

	15:  TON_29(IN:=TRUE , PT:=t#100ms , Q=> , ET=> );
		IF TON_29.Q THEN   iControlWord1:=6;
		TON_14(IN:=FALSE);
		TON_13(IN:=FALSE);
		 step2:=Step2+1; END_IF

	16:	TON_30(IN:=TRUE , PT:=t#100ms , Q=> , ET=> );
		IF TON_30.Q THEN TON_29(IN:=FALSE);  iControlWord1:=7; step2:=Step2+1; END_IF



	17:	TON_13(IN:=TRUE , PT:= T#0.5s, Q=> , ET=> );
		IF TON_13.Q THEN iControlWord1:=15; TON_30(IN:=FALSE);  Step2:=Step2+1; END_IF



	18:	IF statusWord.2 THEN    iControlWord1.4:=TRUE;
		bAServoUpAuto:=FALSE;
		step2:=Step2+1;
		END_IF


	19:	TON_14(IN:=TRUE , PT:= t#2s, Q=> , ET=> );
		IF TON_14.Q THEN  step:=Step+1; END_IF
		step2:=Step2+1;

	20:	IF statusWord.10 THEN
		iControlWord1.4:=FALSE;
		step2:=Step2+1;
		END_IF


	21:	IF bIGripperVerticalHome THEN
		bAPlaceOver:=TRUE;
		step2:=Step2+1;
		END_IF sMessage_Gripper:='  Check Vertical  Home Reed Switch ';


	22:	iControlWord1:=7;
		step2:=Step2+1;

	23:	TON_8(IN:=FALSE);
		TON_9(IN:=FALSE);
		TON_10(IN:=FALSE);
		TON_11(IN:=FALSE);
		TON_12(IN:=FALSE);
		TON_13(IN:=FALSE);
		TON_14(IN:=FALSE);
		TON_29(IN:=FALSE);
		TON_30(IN:=FALSE);
		step2:=Step2+1;

	24:	CountServo:=CountServo+1;
		step2:=Step2+1;

	25:	IF CountServo=3 THEN
		iACountServoToSepUnit:= CountServo;

		step2:=Step2+1;
		ELSIF CountServo<3 THEN
		step2:=Step2+1;
		END_IF

	26:	step2:=0;


END_CASE




IF bAutoModeOn AND CountServo = 0 THEN
iDropPosHmi:=iDropPos1Hmi;

ELSIF bAutoModeOn AND  CountServo=1 THEN
iDropPosHmi:=iDropPos2Hmi;
ELSIF bAutoModeOn AND  CountServo = 2 THEN
iDropPosHmi:=iDropPos3Hmi;
END_IF


iControlWord1.7;

IF  NOT bIEmergencySwitch OR bStopHmi OR bServoOff  OR bIMcStop THEN
iControlWord1:=7;
step:=0;
step2:=0;

bChkEndSensor:=FALSE;
bServoStartedInAuto:=FALSE;
bAServoFwdStart2:=FALSE;
bHomingDone:=FALSE;
bAModeWrite:=FALSE;
diTargetVelocity1:=0;
iControlWord1.4:=FALSE;
bAServoDownDone:=FALSE;
TON_1(IN:=FALSE);
TON_2(IN:=FALSE);
TON_3(IN:=FALSE);
TON_4(IN:=FALSE);
TON_5(IN:=FALSE);
TON_6(IN:=FALSE);
TON_7(IN:=FALSE);
bAServoDown1Done:=FALSE;
bAServoUpAuto:=FALSE;
bAPlaceOver:=FALSE;
bPauseOperationEn1:=FALSE;
bServoReumeActive1:=FALSE;
bServoPauseActive1:=FALSE;
bPauseOperationEn5:=FALSE;
bServoPauseActive5:=FALSE;
bPauseOperationEn3:=FALSE;
bServoPauseActive3:=FALSE;
bServoReumeActive3:=FALSE;
bPauseOperationEn2:=FALSE;
bServoPauseActive2:=FALSE;
 bServoReumeActive2:=FALSE;
bPauseOperationEn6:=FALSE;
bServoPauseActive6:=FALSE;
bServoReumeActive6:=FALSE;
bServoReachedUp:=FALSE;
END_IF

(*==================Pause & Resume Logic for servo after start==================*)


(*===========Pause operation Enable Condition=================*)
IF ( step>0  AND step <= 10 )  THEN
bPauseOperationEn1:=TRUE;
ELSE
bPauseOperationEn1:=FALSE;
bServoReumeActive5:=FALSE;
END_IF


IF bAutoModeOn AND bPauseOperationEn1 AND  bAPauseSeq THEN iControlWord1:=7; bServoPauseActive1:=TRUE; END_IF

IF bServoPauseActive1 AND NOT bAPauseSeq  THEN bServoReumeActive1:=TRUE; ELSE bServoReumeActive1:=FALSE;  END_IF
R_TRIG_1(CLK:= bServoReumeActive1 , Q=> );

IF R_TRIG_1.Q THEN   step:=1; bServoPauseActive1:=FALSE;  END_IF



(*===========Pause operation Enable Condition for return in Pick Side=================*)
IF ( step>=35  AND step <= 37 )AND  bAutoModeOn  THEN
bPauseOperationEn5:=TRUE;
ELSE
bPauseOperationEn5:=FALSE;
END_IF


IF bAutoModeOn AND bPauseOperationEn5 AND  bAPauseSeq THEN iControlWord1:=7; bServoPauseActive5:=TRUE; END_IF

IF bServoPauseActive5 AND NOT bAPauseSeq  THEN bServoReumeActive5:=TRUE; ELSE bServoReumeActive5:=FALSE;  END_IF
R_TRIG_5(CLK:= bServoReumeActive5 , Q=> );


IF R_TRIG_5.Q THEN   step:=28; bServoPauseActive5:=FALSE;  END_IF








(*===========Pause operation Enable Condition for Third Speed=================*)
IF  ( step >= 23 AND  step <=24 )  THEN
bPauseOperationEn3:=TRUE;
ELSE
bPauseOperationEn3:=FALSE;
END_IF



IF bAutoModeOn AND bPauseOperationEn3 AND  bAPauseSeq THEN iControlWord1:=0; bServoPauseActive3:=TRUE; END_IF

IF bServoPauseActive3 AND NOT bAPauseSeq  THEN bServoReumeActive3:=TRUE; ELSE bServoReumeActive3:=FALSE;   END_IF
R_TRIG_3(CLK:= bServoReumeActive3 , Q=> );

IF R_TRIG_3.Q THEN  step:=1; bServoPauseActive3:=FALSE;  END_IF




(*===========Pause operation Enable Condition for Drop Side=================*)
IF  ( step2 >= 0 AND  step2 <=9 )  THEN
bPauseOperationEn2:=TRUE;
ELSE
bPauseOperationEn2:=FALSE;
END_IF



IF bAutoModeOn AND bPauseOperationEn2 AND  bAPauseSeq THEN iControlWord1:=0; bServoPauseActive2:=TRUE;  END_IF

IF bServoPauseActive2 AND NOT bAPauseSeq  THEN bServoReumeActive2:=TRUE;(*ELSE bServoReumeActive2:=FALSE;*)   END_IF
R_TRIG_2(CLK:= bServoReumeActive2 , Q=> );

IF R_TRIG_2.Q AND NOT temp11 THEN  step2:=0; bServoPauseActive2:=FALSE;  bServoReumeActive2:=FALSE;
ELSIF  temp11  AND  R_TRIG_2.Q THEN step2:=4;  bServoPauseActive2:=FALSE; temp11:=FALSE;  bServoReumeActive2:=FALSE;    END_IF



(*===========Pause operation Enable Condition for Drop Side  Return   =================*)
IF  ( step2 >= 19 AND  step2 <=20 )  THEN
bPauseOperationEn6:=TRUE;
ELSE
bPauseOperationEn6:=FALSE;
END_IF



IF bAutoModeOn AND bPauseOperationEn6 AND  bAPauseSeq THEN iControlWord1:=0; bServoPauseActive6:=TRUE;  END_IF

IF bServoPauseActive6 AND NOT bAPauseSeq  THEN bServoReumeActive6:=TRUE;ELSE bServoReumeActive6:=FALSE;   END_IF
R_TRIG_6(CLK:= bServoReumeActive6 , Q=> );

IF R_TRIG_6.Q THEN  step2:=15; bServoPauseActive6:=FALSE;   END_IF
END_PROGRAM

(* POU Auto/Gripper/PickAndPlaceUnit, ST *)
PROGRAM PickAndPlaceUnit
VAR
	step: INT;
	tL_BPistonCloseDly: TON;
	bIGripperVerticalHomeTemp: BOOL;
	test: BOOL;
	bAServoDownDone1: BOOL;
	TON_1: TON;
	bIConeEjectionPistonEndtemp: BOOL;
	bIConeEjectionPistonHomeTemp: BOOL;
	Timer1: TON;
	Timer2: TON;
	SepHoriCylHomeRsErrChk: RS_Error;
	SepHoriCylHomeRsErr: BOOL;
	SepHoriCylEndRsErrChk: RS_Error;
	SepHoriCylEndRsErr: BOOL;
END_VAR
	IF NOT  bIEmergencySwitch OR   bStopHmi OR bServoOff OR bIMcStop THEN
	tL_BPistonCloseDly(IN:=FALSE);
	Timer2(IN:=FALSE);
	step:=0;
	bQASeparatorHorizontalPistonValveREV:=FALSE;
	bQALengthTightPistonValve:=FALSE;
	bQABreadthTightPistonValve:=FALSE;
	 bAConePickDone:=FALSE;
	bAServoDownDone:=FALSE;
	Timer1(IN:=FALSE);
	bQASeparatorHorizontalPistonValveFWD:=FALSE;
	TON_1(IN:=FALSE);
	bAServoFwdStart2:=FALSE;
	bQAConeEjectionPistonValve:=FALSE;
	bAServoDown1Done:=FALSE;
	bAServoUpAuto:=FALSE;
	bServoReachedUp:=FALSE;
	bAPlaceOver:=FALSE;
END_IF


CASE step OF

	0:	tL_BPistonCloseDly(IN:=FALSE);
		Timer2(IN:=FALSE);
		 step:=step+1;

	1:	 step:=step+1;

	2:	IF bAutoModeOn AND bAServoDownDone (*AND bILengthTightPistonHome*) AND bIBreadthTightPistonHome THEN
		tL_BPistonCloseDly(IN:=TRUE , PT:=T#0.2s , Q=> , ET=> );
		IF tL_BPistonCloseDly.Q THEN   step:=step+1;END_IF
		END_IF

	3:	 step:=step+1;

	4:	IF bAutoModeOn AND bAServoDownDone (*AND bILengthTightPistonHome*) AND bIGripperVerticalEnd   AND bIBreadthTightPistonHome
		AND  NOT bAPauseSeq  AND NOT bAL_BTightHomeSenRsError THEN
		bQASeparatorHorizontalPistonValveREV:=FALSE;
		bQALengthTightPistonValve:=TRUE;
		bQABreadthTightPistonValve:=TRUE;
		 step:=step+1;
		END_IF

	5:	Timer2(IN:=TRUE , PT:=t#2s , Q=> , ET=> );bAServoDownDone:=FALSE;
		IF Timer2.Q THEN  bAConePickDone:=TRUE; step:=step+1; END_IF

	6:	IF bAutoModeOn AND bIGripperVerticalHome AND bServoReachedUp AND bISeparatorHorizontalPistonEnd  AND bISeparatorVerticalPistonHome
		 AND (bACartonReady_23 OR bACartonReady_24) AND  NOT bAPauseSeq  AND NOT bIGripperVerticalEnd THEN
		bQASeparatorHorizontalPistonValveFWD:=TRUE;
		TON_1(IN:=FALSE);
		Timer2(IN:=FALSE);
		tL_BPistonCloseDly(IN:=FALSE);
		step:=step+1;
		END_IF

	7:	 step:=step+1;

	8:	IF  bAutoModeOn  AND bISeparatorHorizontalPistonHome  AND NOT bHmiColourChangeBit2_24 AND NOT bASepaHoriForwdEndRsError  AND NOT SeparatorAlertbit THEN

		(*bACartonReady_24:=FALSE;*)
		bServoReachedUp:=FALSE;
		TON_1(IN:=TRUE , PT:=t#0.3s  , Q=> , ET=> );
		IF TON_1.Q THEN step:=step+1; END_IF
		END_IF

	9:	 step:=step+1;

	10:	IF NOT bAPauseSeq THEN bAServoFwdStart2:=TRUE;
		 step:=step+1;
		END_IF

	11:	 step:=step+1;

	12:	IF  bAutoModeOn  AND bISeparatorHorizontalPistonHome  AND bAServoDown1Done  AND NOT bAPauseSeq THEN
		bQALengthTightPistonValve:=FALSE;

		step:=step+1;
		END_IF

	13:	 step:=step+1;

	14:	IF  bAutoModeOn AND bIConeEjectionPistonHome AND NOT bAPauseSeq  THEN
		bQAConeEjectionPistonValve:=TRUE;
		bAServoDown1Done:=FALSE;
		step:=step+1;
		END_IF

	15:	timer1(IN:=TRUE , PT:=T#0.5s , Q=> , ET=> );
		IF  timer1.Q   THEN step:=step+1; END_IF

	16:	IF  bAutoModeOn  THEN

		bAServoUpAuto:=TRUE;
		step:=step+1;
		END_IF

	17:	 step:=step+1;

	18:	IF bAutoModeOn AND  bIGripperVerticalHome (*AND statusWord.10  *)THEN
		bQABreadthTightPistonValve:=FALSE;
		bQASeparatorHorizontalPistonValveFWD:=FALSE;
		step:=step+1;
		END_IF

	19:	 step:=step+1;

	20:	 IF bIBreadthTightPistonHome(* AND bILengthTightPistonHome*)  AND NOT bAPauseSeq  AND NOT bAL_BTightHomeSenRsError  THEN
		 bQAConeEjectionPistonValve:=FALSE;
		step:=step+1;
		END_IF

	21:	 step:=step+1;

	22:	IF bAPlaceOver AND bIGripperVerticalHome  AND bISeparatorVerticalPistonHome AND NOT bAPauseSeq  THEN
		bQASeparatorHorizontalPistonValveREV:=TRUE;
		step:=step+1;
		END_IF

	23:	step:=step+1;

	24:	IF bISeparatorHorizontalPistonEnd  AND NOT bASepaHoriRevValveRsError THEN

		bAPlaceOver:=FALSE;
		step:=0;
		END_IF

END_CASE
END_PROGRAM

(* POU FunctionBlocks/RS_Error, ST *)
FUNCTION_BLOCK RS_Error
VAR_INPUT
	bValveOutOn: BOOL;
	bReedSwithIn: BOOL;
	bErroReset: BOOL;
	sMsgIn: STRING;
	RS_ErrChkDly: TIME;
END_VAR
VAR_OUTPUT
	bRsError: BOOL;
	sMsgOut: STRING;
END_VAR
VAR
	FbStep: INT;
	Timer1: TON;
END_VAR
CASE FbStep OF


	0:	Timer1(IN:=FALSE); FbStep:=FbStep+1;

	1:	IF bValveOutOn THEN FbStep:=FbStep+1; END_IF

	2:	Timer1(IN:=TRUE , PT:=RS_ErrChkDly , Q=> , ET=> );
		IF Timer1.Q THEN FbStep:=FbStep+1;
		ELSIF NOT  Timer1.Q AND bReedSwithIn THEN  FbStep:=0; END_IF

	3:	IF bReedSwithIn THEN  FbStep:=FbStep+1;
		ELSIF NOT bReedSwithIn THEN FbStep:=FbStep+2; END_IF

	4:	IF  NOT bValveOutOn THEN sMsgOut:=sMsgIn;  FbStep:=0; END_IF

	5:	bRsError:=TRUE; FbStep:=FbStep+1;

	6:	IF   bReedSwithIn AND   bErroReset THEN bRsError:=FALSE; sMsgOut:='' ;  FbStep:=0;
		ELSIF   NOT bReedSwithIn AND   bRsError  AND  bErroReset THEN bRsError:=FALSE;   sMsgOut:='' ;   FbStep:=0;
		 END_IF

END_CASE
END_FUNCTION_BLOCK

(* POU Auto1/DataLog/DataLog_1, ST *)
PROGRAM DataLog_1
VAR
	stStation1_ProductionData: Production_Data;
	ST1_ProductionDataValues: STRING(3000);
	S1_iCyc_Count_DISP: INT;
	S1_iACT_HLD_TIMEDISP: INT;
	stActiveuserCredential: BOOL;
	nPressureMaxvalue: REAL;
	OperatorName: STRING;
	nMinimumTopTempLimit_ST1: INT;
	nMaximumTopTempLimit_ST1: INT;
	nTOPTempMaxvalue: UINT;
	nMinimumBTMTempLimit_ST1: INT;
	nBTMTempMaxvalue: UINT;
	nMaximumBTMTempLimit_ST1: INT;
	Set_HLDTIME: INT;
	S_1_iPressure: REAL;
	rS_PressureRange1: REAL;
	nMaxEnergy: REAL;
	nMaxPower: REAL;
	S_iSET_COUNT: INT;
	S1_iTotCyc_Count_DISP: INT;
	sJobStatus_ST1: STRING;
	sStation1_ProductionData_FileName: STRING(80) := 'Hard Disk\Reports\Test1\ProductionData.csv';
	Fb_LoagProductionData: DATA_LOG_Save;
	SaveData: BOOL;
	ST1_ProductionData: STRING(500);
	Fb_CreateFileFormat_1: Fb_CreateFileFormat;
	bEnableFileFormat: BOOL;
	wTodayTemp: STRING;
	sDateTemp: STRING;
	sOLDFileName_ST1: T_MaxString;
	Fb_FormatDrive_1: Fb_FormatDrive;
	bFileDelete: BOOL;
	Fb_CopyBackupAL_Server_LogOf_1: Fb_CopyFileToRemotePC;
	bool2: BOOL;
	bAstart: BOOL;
	TON_1: TON;
	TON_2: TON;
	CTU_1: CTU;
	R_TRIG_1: R_TRIG;
	R_TRIG_2: R_TRIG;
	bACreateNewFile: BOOL;
	ReportStep: INT;
	bANewDay: BOOL;
	Timer1: TON;
	Timer2: TON;
	R_TRIG1: R_TRIG;


	iUnitBNetWtTemp1: REAL;
	rRetUnitBWeightTemp1: REAL;
	StepTemp1: INT;
	rRetUnitBWeightTemp2: REAL;
	StepTemp2: INT;
	BCreateDir: BOOL;
	FB_CreateDir_1: FB_CreateDir;
	bANewDaytemp: BOOL;
	bit2: BOOL;
	hfile: UINT;
	FB_FileOpen_1: FB_FileOpen;
	test: BOOL;
	bit3: BOOL;
	FB_FileWrite_1: FB_FileWrite;
	bEnableFileFormattemp: BOOL;
	BDelete: BOOL;
	FB_FileDelete_1: FB_FileDelete;
	Timer3: TON;
	iCartoNoHmiTemp: DWORD;
	dateInint: WORD;
	E_OpenPath: E_OpenPath;
	FB_FileDelete_2: FB_FileDelete;
END_VAR
FileCreateTemp;

Fb_CreateFileFormat_1(
	sInputMessage:=ST1_ProductionData ,
	sFileName:='ProductionData' ,
	sDirectory:= '\\WELCOME-PC\Reports\' (*  'Hard Disk\Reports\Indo\'  *) ,
	bEnable:=bEnableFileFormat ,
	wToday:=wTodayTemp ,
	sDate=> sDateTemp,
	bNewDateFound=> bANewDay,
	sOldFileName=>sOLDFileName_ST1 ,
	sFilePathFinal=> );

FB_FileDelete_2(
	sNetId:='127.255.255.1.1.1' ,
	sPathName:= sStation1_ProductionData_FileName ,
	ePath:=E_OpenPath ,
	bExecute:=bFileDelete ,
	tTimeout:=t#1s ,
	bBusy=> ,
	bError=> ,
	nErrId=> );


bLoadPgm;
IF (bloadRecipeHmi OR bSaveRecipeHmi) THEN
iCartoNoHmiTemp:=iCartoNoHmi;
ELSE
iCartoNoHmiTemp:=(ITotalSample +iCartoNoHmi);
END_IF

iCartonSample:=iCartoNoHmiTemp;

		stStation1_ProductionData.S_No						:=INT_TO_STRING( Pgm_NoHmi );
		stStation1_ProductionData.CartonNo					:=DWORD_TO_STRING(iCartoNoHmiTemp);
		stStation1_ProductionData.SDateF					:= (sDATEFinal);
		stStation1_ProductionData.sShift						:=(sShitToReport);
	(*	stStation1_ProductionData.ActualNetWt				:=REAL_TO_STRING(rRetUnitAWeight); *)
		stStation1_ProductionData.LotNo					:=DWORD_TO_STRING(iLotNoHmi);
		stStation1_ProductionData.sCount					:=(iCountHmi);
		stStation1_ProductionData.NetWt					:=REAL_TO_STRING(var_5);
		stStation1_ProductionData.StandardGrossWt			:=(var_7);
		stStation1_ProductionData.sTolerance				:=REAL_TO_STRING(NetToleranceHmi);
		stStation1_ProductionData.sEmpConeWt				:=REAL_TO_STRING(iWeightHmi);




		(*	######## LOG PRODUCTION DATA		#####	*)

ST1_ProductionDataValues:= CONCAT(stStation1_ProductionData.S_No,',');
ST1_ProductionDataValues:=	 CONCAT( ST1_ProductionDataValues,stStation1_ProductionData.CartonNo);
ST1_ProductionDataValues:= CONCAT( ST1_ProductionDataValues,',');
ST1_ProductionDataValues:=	 CONCAT( ST1_ProductionDataValues,stStation1_ProductionData.SDateF	);
ST1_ProductionDataValues:= CONCAT( ST1_ProductionDataValues,',');
ST1_ProductionDataValues:=	 CONCAT( ST1_ProductionDataValues,stStation1_ProductionData.sShift	);
ST1_ProductionDataValues:= CONCAT( ST1_ProductionDataValues,',');
(*ST1_ProductionDataValues:=	 CONCAT( ST1_ProductionDataValues,stStation1_ProductionData.ActualNetWt	);
ST1_ProductionDataValues:= CONCAT( ST1_ProductionDataValues,',');*)
ST1_ProductionDataValues:=	 CONCAT( ST1_ProductionDataValues,stStation1_ProductionData.LotNo);
ST1_ProductionDataValues:= CONCAT( ST1_ProductionDataValues,',');
ST1_ProductionDataValues:=	 CONCAT( ST1_ProductionDataValues,stStation1_ProductionData.sCount);
ST1_ProductionDataValues:= CONCAT( ST1_ProductionDataValues,',');
ST1_ProductionDataValues:=	 CONCAT( ST1_ProductionDataValues,stStation1_ProductionData. NetWt );
ST1_ProductionDataValues:= CONCAT( ST1_ProductionDataValues,',');
ST1_ProductionDataValues:=	 CONCAT( ST1_ProductionDataValues,stStation1_ProductionData.StandardGrossWt);
ST1_ProductionDataValues:= CONCAT( ST1_ProductionDataValues,',');
ST1_ProductionDataValues:=	 CONCAT( ST1_ProductionDataValues,stStation1_ProductionData.sEmpConeWt);
ST1_ProductionDataValues:= CONCAT( ST1_ProductionDataValues,'$0A');     (**)

(*==========Saving the Data to Report===========*)

sStation1_ProductionData_FileName:= Fb_CreateFileFormat_1.sOldFileName ; (*    'Hard Disk\Reports\Test1\ProductionData.csv' ;*)


Fb_LoagProductionData(
	bStartDataLog:= SaveData ,
	sDataLogFileName:=sStation1_ProductionData_FileName ,
	LogData:=ST1_ProductionDataValues ,
	bErrorDataLog=> );






(*=============== file copy from CX Controller to Remote PC & File Delete In CX Device======================*)


	Fb_CopyBackupAL_Server_LogOf_1(
		bMakeDirectory:= ,
		bCopyFile:=bool2,
		sDestDriveName:= '\\WELCOME-PC\Reports\   ' ,
		sSourceDirectory:='\Hard Disk\Reports\Indo' ,
		 );

(*\\ramrajg-nb2\Ramaraj_public\   *)

  (*Hard Disk\Reports\  *)

Fb_FormatDrive_1(sDriveName:='\\WELCOME-PC\Reports\' , bFormatDisk:=bFileDelete );


CASE ReportStep OF

	0:	 IF R_TRIG1.Q   THEN  FileCreateTemp:=TRUE; Timer3(IN:=FALSE); ReportStep:=1; END_IF

	1:	(*		##### Station 1 Production Data	#####	*)

		ST1_ProductionData:= CONCAT( 'Prg No',',');
		ST1_ProductionData:=	 CONCAT( ST1_ProductionData,'Carton No');
		ST1_ProductionData:= CONCAT( ST1_ProductionData,',');
		ST1_ProductionData:=	 CONCAT( ST1_ProductionData,'Date');
		ST1_ProductionData:= CONCAT( ST1_ProductionData,',');
		ST1_ProductionData:=	 CONCAT( ST1_ProductionData,'Shift');
		ST1_ProductionData:= CONCAT( ST1_ProductionData,',');
	(*	ST1_ProductionData:=	 CONCAT( ST1_ProductionData,'Unit');
		ST1_ProductionData:= CONCAT( ST1_ProductionData,',');*)
		ST1_ProductionData:=	 CONCAT( ST1_ProductionData,'Lot No');
		ST1_ProductionData:= CONCAT( ST1_ProductionData,',');
		ST1_ProductionData:=	 CONCAT( ST1_ProductionData,'Count');
		ST1_ProductionData:= CONCAT( ST1_ProductionData,',');
		ST1_ProductionData:=	 CONCAT( ST1_ProductionData,'Net Weight');
		ST1_ProductionData:= CONCAT( ST1_ProductionData,',');
		ST1_ProductionData:=	 CONCAT( ST1_ProductionData,'Gross Weight');
		ST1_ProductionData:= CONCAT( ST1_ProductionData,',');
		ST1_ProductionData:=	 CONCAT( ST1_ProductionData,'Tolerance');
		ST1_ProductionData:= CONCAT( ST1_ProductionData,',');
		ST1_ProductionData:=	 CONCAT( ST1_ProductionData,' Empty Cone Weight');
		ST1_ProductionData:= CONCAT( ST1_ProductionData,'$0A');

		ReportStep:=2;

	2:	Timer1(IN:=FALSE);
		bANewDay:=FALSE;
		ReportStep:=3;


	3:	bEnableFileFormat:=TRUE;
		Timer1(IN:=TRUE , PT:=T#100ms , Q=> , ET=> );
		IF Timer1.Q THEN bEnableFileFormat:=FALSE;  ReportStep:=4; END_IF


	4:	(*IF R_TRIG1.Q THEN  *)
		SaveData:=TRUE;
		Timer1(IN:=FALSE);
		ReportStep:=5;

	5:	Timer3(IN:=TRUE , PT:=T#20s , Q=> , ET=> );
		IF Timer3.Q THEN SaveData:=FALSE;bFileDelete:=TRUE;  ReportStep:=6; END_IF

	6:	 bFileDelete:=FALSE;Timer3(IN:=FALSE); FileCreateTemp:=FALSE; ReportStep:=0;

END_CASE



R_TRIG1(CLK:=bACyclePass , Q=> );


CASE StepTemp1 OF
	0:	IF bRetUnitBStart THEN rRetUnitBWeightTemp1:=rRetUnitBWeight; StepTemp1:=StepTemp1+1; END_IF

	1:	IF UnitBCompleteCheckCount.CV = 18 AND bAutoModeOn THEN rRetUnitBWeightTemp2:=rRetUnitBWeightTemp1;  StepTemp1:=0; END_IF
 END_CASE




CASE StepTemp2 OF
	0:	IF bRetUnitBStart THEN rRetUnitBWeightTemp1:=rRetUnitBWeight; StepTemp2:=StepTemp2+1; END_IF

	1:	IF c18_ConeCounter1.CV = 18 AND bAutoModeOn THEN rRetUnitBWeightTemp2:=rRetUnitBWeightTemp1; c18_ConeCounter1.RESET:=TRUE;  StepTemp2:=StepTemp2+1; END_IF

	2:	c18_ConeCounter1.RESET:=FALSE;  StepTemp2:=0;
 END_CASE
END_PROGRAM

(* POU FunctionBlocks/DATA_LOG_Save, ST *)
FUNCTION_BLOCK DATA_LOG_Save
VAR_INPUT
	bStartDataLog: BOOL;
	sDataLogFileName: STRING;
	LogData: STRING(1024);

END_VAR
VAR_OUTPUT

	bErrorDataLog: BOOL;
END_VAR
VAR

	R_TRIGStartDataLog: R_TRIG;
	nstep: INT;

	FB_OpenFile_Datalog: FB_FileOpen;
	nFB_OpenFile_Datalog_Errid: UDINT;

	FB_WriteFile_Datalog: FB_FileWrite;
	nFB_WriteFile_Datalog_ErrId: UDINT;

	FB_CloseFile_Datalog: FB_FileClose;
	nFB_CloseFile_Datalog_ErrId: UDINT;
	hDataLogSrcFile: UINT;

END_VAR
R_TRIGStartDataLog(CLK:=bStartDataLog , Q=> );
IF R_TRIGStartDataLog.Q THEN
		nstep :=1;
	END_IF

CASE nstep OF

	0:
		;
		FB_OpenFile_Datalog.bExecute:=FALSE;
		FB_WriteFile_Datalog.bExecute:=FALSE;
		FB_CloseFile_Datalog.bExecute:=FALSE;

	1:		(* do nothing *)
			nstep:=nstep+1;

	2:		(* ####	File Open ####*)

			FB_OpenFile_Datalog(  bExecute := FALSE  );
			FB_OpenFile_Datalog(	sNetId :='127.255.255.1.1.1' ,
			sPathName := sDataLogFileName,
			nMode := FOPEN_MODEAPPEND    ,
			ePath := PATH_GENERIC,
			tTimeout := T#2s,
			bExecute := TRUE );
			nstep := nstep+ 1;



	3:		FB_OpenFile_Datalog( bExecute := FALSE );
			IF ( NOT FB_OpenFile_Datalog.bBusy ) THEN
			IF ( FB_OpenFile_Datalog.bError ) THEN
			nFB_OpenFile_Datalog_Errid := FB_OpenFile_Datalog.nErrId;
			bErrorDataLog := TRUE;
			nstep := 50;
			ELSE
			hDataLogSrcFile := FB_OpenFile_Datalog.hFile;
			nstep := nstep + 1;
			END_IF
			END_IF

	4:		(*write data to destination file*)
			(*num:=num+1;*)
			FB_WriteFile_Datalog( bExecute := FALSE );
			FB_WriteFile_Datalog(	sNetId:='127.255.255.1.1.1',
			hFile:=FB_OpenFile_Datalog.hFile,
			pWriteBuff:= ADR(LogData),
			cbWriteLen:= LEN(LogData),		(*	i_len,	*)
			bExecute:=TRUE,
			tTimeout:=T#2s );
			nstep := nstep + 1;

	5:		FB_WriteFile_Datalog( bExecute := FALSE );
			IF ( NOT FB_WriteFile_Datalog.bBusy ) THEN
			IF ( FB_WriteFile_Datalog.bError ) THEN
			nFB_WriteFile_Datalog_ErrId := FB_WriteFile_Datalog.nErrId;
			bErrorDataLog := TRUE;
			nstep := 50;
			ELSE
			hDataLogSrcFile := FB_OpenFile_Datalog.hFile;
			nstep := nstep + 1;
			END_IF
			END_IF

	6:		(* close the destination file *)
			FB_CloseFile_Datalog( bExecute := FALSE );
			FB_CloseFile_Datalog( 	sNetId:='127.255.255.1.1.1' ,
			hFile:=FB_OpenFile_Datalog.hFile,
			bExecute:=TRUE,
			tTimeout:=T#2s );
			nstep := nstep + 1;

	7:		FB_CloseFile_Datalog( bExecute := FALSE );
			IF ( NOT FB_CloseFile_Datalog.bBusy ) THEN
			IF ( FB_CloseFile_Datalog.bError ) THEN
			nFB_CloseFile_Datalog_ErrId := FB_CloseFile_Datalog.nErrId;
			bErrorDataLog := TRUE;
			END_IF
			nstep := 0;
			END_IF

END_CASE
END_FUNCTION_BLOCK

(* POU FunctionBlocks/Fb_CreateFileFormat, LD *)
FUNCTION_BLOCK Fb_CreateFileFormat
VAR
	Fb_OpenFile: FB_FileOpen;
	Fb_WriteFile: FB_FileWrite;
	F_Trig1: F_TRIG;
	F_Trig2: F_TRIG;
	Fb_closeFile: FB_FileClose;
	F_Trig3: F_TRIG;


	SysteMtime: FB_LocalSystemTime;
	stSystemtimeAlrm: Timestruct;

	sFileName_Temp: T_MaxString;


	bCreateFileTrig: R_TRIG;
	bCreateFile: BOOL;
	Fb_SavePersistant: FB_WritePersistentData;
	TuneparaSave: BOOL;
END_VAR
VAR_INPUT

	sInputMessage: STRING(255);
	sFileName: T_MaxString;
	sDirectory: T_MaxString;
	bEnable: BOOL;

END_VAR
VAR_OUTPUT

	sDate: STRING;

	bNewDateFound: BOOL;
END_VAR

VAR_OUTPUT PERSISTENT
	sOldFileName: T_MaxString;
	sFilePathFinal: t_MaxString;
END_VAR
VAR PERSISTENT
	sOldDate: STRING;
	sNewFileName_Temp: T_MaxString;
END_VAR
VAR_IN_OUT PERSISTENT
	wToday: STRING;
END_VAR
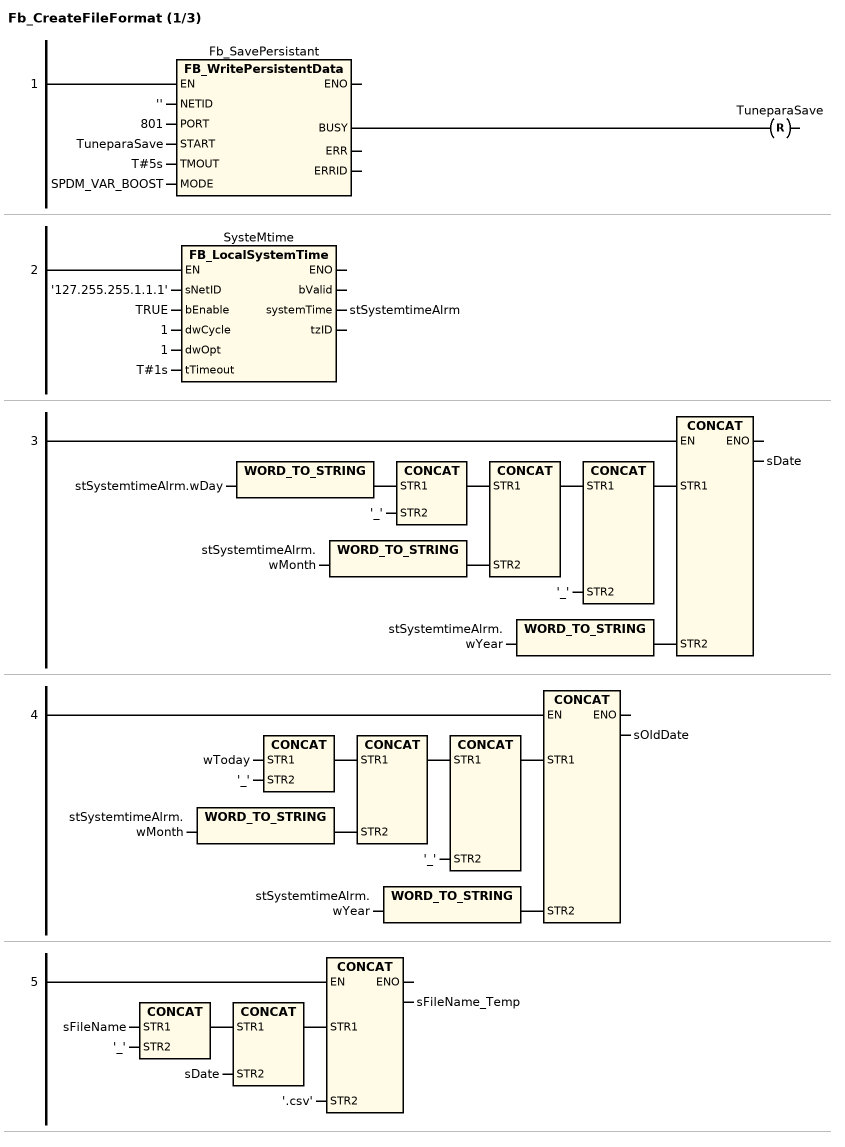
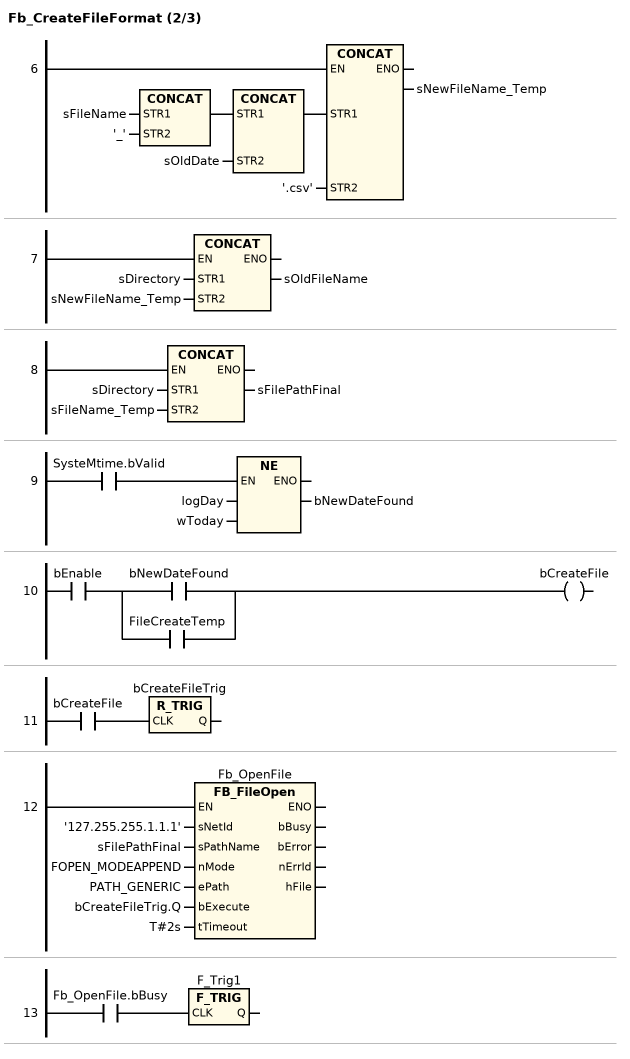
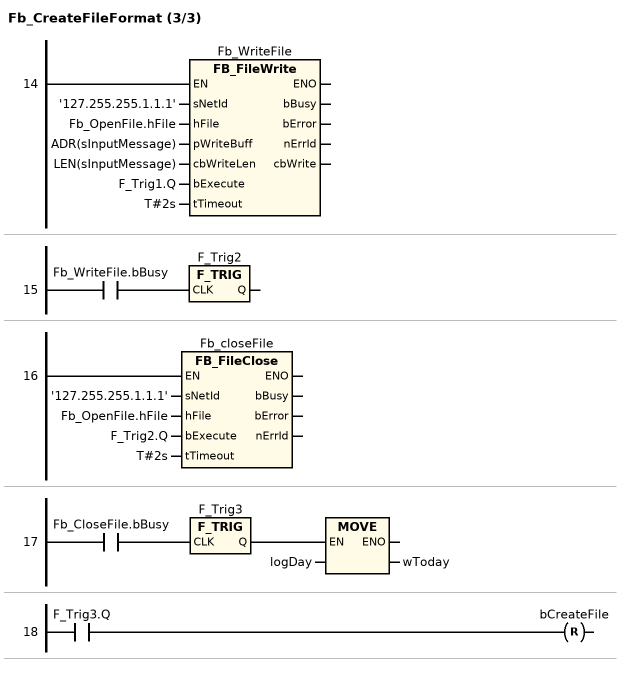
_LD_ (* Ladder Diagram *)
NETWORK 1
	*
		EN --- Fb_SavePersistant:FB_WritePersistentData(NETID: '', PORT: 801, START: TuneparaSave, TMOUT: T#5s, MODE: SPDM_VAR_BOOST) => R TuneparaSave
NETWORK 2
	*
		EN --- SysteMtime:FB_LocalSystemTime(sNetID: '127.255.255.1.1.1', bEnable: TRUE, dwCycle: 1, dwOpt: 1, tTimeout: T#1s, systemTime => stSystemtimeAlrm)
NETWORK 3
	*
		EN --- CONCAT(STR1: CONCAT(STR1: CONCAT(STR1: CONCAT(STR1: WORD_TO_STRING(stSystemtimeAlrm.wDay), STR2: '_'), STR2: WORD_TO_STRING(stSystemtimeAlrm.wMonth)), STR2: '_'), STR2: WORD_TO_STRING(stSystemtimeAlrm.wYear)) => sDate
NETWORK 4
	*
		EN --- CONCAT(STR1: CONCAT(STR1: CONCAT(STR1: CONCAT(STR1: wToday, STR2: '_'), STR2: WORD_TO_STRING(stSystemtimeAlrm.wMonth)), STR2: '_'), STR2: WORD_TO_STRING(stSystemtimeAlrm.wYear)) => sOldDate
NETWORK 5
	*
		EN --- CONCAT(STR1: CONCAT(STR1: CONCAT(STR1: sFileName, STR2: '_'), STR2: sDate), STR2: '.csv') => sFileName_Temp
NETWORK 6
	*
		EN --- CONCAT(STR1: CONCAT(STR1: CONCAT(STR1: sFileName, STR2: '_'), STR2: sOldDate), STR2: '.csv') => sNewFileName_Temp
NETWORK 7
	*
		EN --- CONCAT(STR1: sDirectory, STR2: sNewFileName_Temp) => sOldFileName
NETWORK 8
	*
		EN --- CONCAT(STR1: sDirectory, STR2: sFileName_Temp) => sFilePathFinal
NETWORK 9
	[SysteMtime.bValid]
		EN --- NE(logDay, wToday) => bNewDateFound
NETWORK 10
	[bEnable] - { [bNewDateFound] | [FileCreateTemp] } --- (bCreateFile)
NETWORK 11
	[bCreateFile] - bCreateFileTrig:R_TRIG(CLK: *)
NETWORK 12
	*
		EN --- Fb_OpenFile:FB_FileOpen(sNetId: '127.255.255.1.1.1', sPathName: sFilePathFinal, nMode: FOPEN_MODEAPPEND, ePath: PATH_GENERIC, bExecute: bCreateFileTrig.Q, tTimeout: T#2s)
NETWORK 13
	[Fb_OpenFile.bBusy] - F_Trig1:F_TRIG(CLK: *)
NETWORK 14
	*
		EN --- Fb_WriteFile:FB_FileWrite(sNetId: '127.255.255.1.1.1', hFile: Fb_OpenFile.hFile, pWriteBuff: ADR(sInputMessage), cbWriteLen: LEN(sInputMessage), bExecute: F_Trig1.Q, tTimeout: T#2s)
NETWORK 15
	[Fb_WriteFile.bBusy] - F_Trig2:F_TRIG(CLK: *)
NETWORK 16
	*
		EN --- Fb_closeFile:FB_FileClose(sNetId: '127.255.255.1.1.1', hFile: Fb_OpenFile.hFile, bExecute: F_Trig2.Q, tTimeout: T#2s)
NETWORK 17
	[Fb_CloseFile.bBusy] - F_Trig3:F_TRIG(CLK: *)
		EN --- MOVE(logDay) => wToday
NETWORK 18
	[F_Trig3.Q] --- (R bCreateFile)
_END_LD_
(* the same logic as Structured Text *)
(* Network 1 *)
Fb_SavePersistant(NETID := '', PORT := 801, START := TuneparaSave, TMOUT := T#5s, MODE := SPDM_VAR_BOOST);
IF Fb_SavePersistant.BUSY THEN TuneparaSave := FALSE; END_IF;
(* Network 2 *)
SysteMtime(sNetID := '127.255.255.1.1.1', bEnable := TRUE, dwCycle := 1, dwOpt := 1, tTimeout := T#1s);
stSystemtimeAlrm := SysteMtime.systemTime;
(* Network 3 *)
sDate := CONCAT(CONCAT(CONCAT(CONCAT(WORD_TO_STRING(stSystemtimeAlrm.wDay), '_'), WORD_TO_STRING(stSystemtimeAlrm.wMonth)), '_'), WORD_TO_STRING(stSystemtimeAlrm.wYear));
(* Network 4 *)
sOldDate := CONCAT(CONCAT(CONCAT(CONCAT(wToday, '_'), WORD_TO_STRING(stSystemtimeAlrm.wMonth)), '_'), WORD_TO_STRING(stSystemtimeAlrm.wYear));
(* Network 5 *)
sFileName_Temp := CONCAT(CONCAT(CONCAT(sFileName, '_'), sDate), '.csv');
(* Network 6 *)
sNewFileName_Temp := CONCAT(CONCAT(CONCAT(sFileName, '_'), sOldDate), '.csv');
(* Network 7 *)
sOldFileName := CONCAT(sDirectory, sNewFileName_Temp);
(* Network 8 *)
sFilePathFinal := CONCAT(sDirectory, sFileName_Temp);
(* Network 9 *)
IF SysteMtime.bValid THEN
	bNewDateFound := logDay <> wToday;
END_IF;
(* Network 10 *)
bCreateFile := bEnable AND (bNewDateFound OR FileCreateTemp);
(* Network 11 *)
bCreateFileTrig(CLK := bCreateFile);
(* Network 12 *)
Fb_OpenFile(sNetId := '127.255.255.1.1.1', sPathName := sFilePathFinal, nMode := FOPEN_MODEAPPEND, ePath := PATH_GENERIC, bExecute := bCreateFileTrig.Q, tTimeout := T#2s);
(* Network 13 *)
F_Trig1(CLK := Fb_OpenFile.bBusy);
(* Network 14 *)
Fb_WriteFile(sNetId := '127.255.255.1.1.1', hFile := Fb_OpenFile.hFile, pWriteBuff := ADR(sInputMessage), cbWriteLen := LEN(sInputMessage), bExecute := F_Trig1.Q, tTimeout := T#2s);
(* Network 15 *)
F_Trig2(CLK := Fb_WriteFile.bBusy);
(* Network 16 *)
Fb_closeFile(sNetId := '127.255.255.1.1.1', hFile := Fb_OpenFile.hFile, bExecute := F_Trig2.Q, tTimeout := T#2s);
(* Network 17 *)
F_Trig3(CLK := Fb_CloseFile.bBusy);
IF F_Trig3.Q THEN
	wToday := logDay;
END_IF;
(* Network 18 *)
IF F_Trig3.Q THEN bCreateFile := FALSE; END_IF;
END_FUNCTION_BLOCK

(* POU FunctionBlocks/Fb_FormatDrive, FBD *)
FUNCTION_BLOCK Fb_FormatDrive
VAR_INPUT
	sDriveName: T_MaxString;
	bFormatDisk: BOOL;
END_VAR
VAR_OUTPUT
END_VAR
VAR
	sDeleteCommand_Temp: T_MaxString;
	sDeleteCommand: T_MaxString;
	nDirectoryLength: INT;
	sFormatedDirectory: T_MaxString;
	FbFormatDisk: NT_StartProcess;
END_VAR
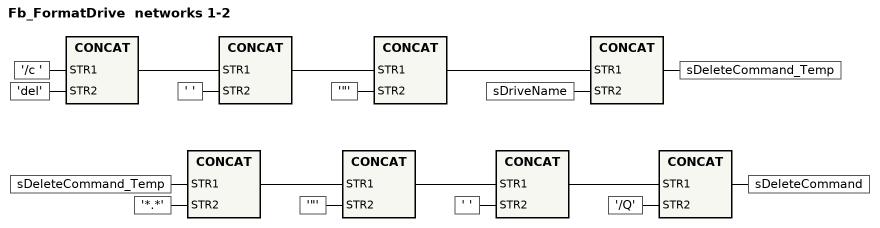
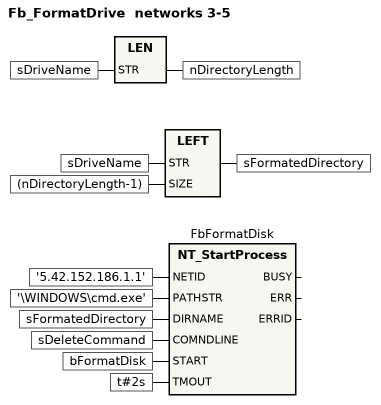
_FBD_ (* Function Block Diagram *)
NETWORK 1
	CONCAT(STR1: CONCAT(STR1: CONCAT(STR1: CONCAT(STR1: '/c ', STR2: 'del'), STR2: ' '), STR2: '"'), STR2: sDriveName) => sDeleteCommand_Temp
NETWORK 2
	CONCAT(STR1: CONCAT(STR1: CONCAT(STR1: CONCAT(STR1: sDeleteCommand_Temp, STR2: '*.*'), STR2: '"'), STR2: ' '), STR2: '/Q') => sDeleteCommand
NETWORK 3
	LEN(STR: sDriveName) => nDirectoryLength
NETWORK 4
	LEFT(STR: sDriveName, SIZE: (nDirectoryLength-1)) => sFormatedDirectory
NETWORK 5
	FbFormatDisk:NT_StartProcess(NETID: '5.42.152.186.1.1', PATHSTR: '\WINDOWS\cmd.exe', DIRNAME: sFormatedDirectory, COMNDLINE: sDeleteCommand, START: bFormatDisk, TMOUT: t#2s)
_END_FBD_
(* the same logic as Structured Text *)
(* Network 1 *)
sDeleteCommand_Temp := CONCAT(CONCAT(CONCAT(CONCAT('/c ', 'del'), ' '), '"'), sDriveName);
(* Network 2 *)
sDeleteCommand := CONCAT(CONCAT(CONCAT(CONCAT(sDeleteCommand_Temp, '*.*'), '"'), ' '), '/Q');
(* Network 3 *)
nDirectoryLength := LEN(sDriveName);
(* Network 4 *)
sFormatedDirectory := LEFT(sDriveName, (nDirectoryLength-1));
(* Network 5 *)
FbFormatDisk(NETID := '5.42.152.186.1.1', PATHSTR := '\WINDOWS\cmd.exe', DIRNAME := sFormatedDirectory, COMNDLINE := sDeleteCommand, START := bFormatDisk, TMOUT := t#2s);
END_FUNCTION_BLOCK

(* POU FunctionBlocks/Fb_CopyFileToRemotePC, FBD *)
FUNCTION_BLOCK Fb_CopyFileToRemotePC
VAR
	sCopyFileCommandTemp: T_MaxString;
	sFormatedDestDirectory: T_Maxstring;
	sCopyFileCommand: T_MaxString;
	sFormatedDirectory: T_MaxString;
	sMakeDirCommand: T_MaxString;

	Fb_SystemTime: FB_LocalSystemTime;
	FB_MakeDirectory: NT_StartProcess;
	Fb_CopyFiles: NT_StartProcess;
END_VAR
VAR_INPUT

	bMakeDirectory: BOOL;
	bCopyFile: BOOL;
	sDestDriveName: T_MaxString;
	sSourceDirectory: T_MaxString;
END_VAR
VAR_OUTPUT
	sFinalDestDirectory: T_MaxString;
END_VAR
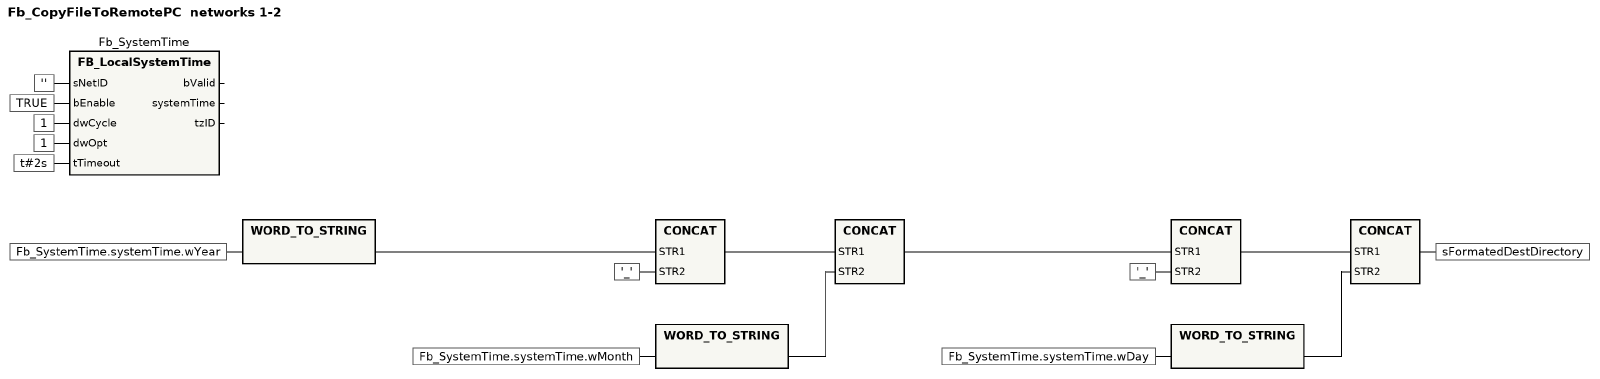
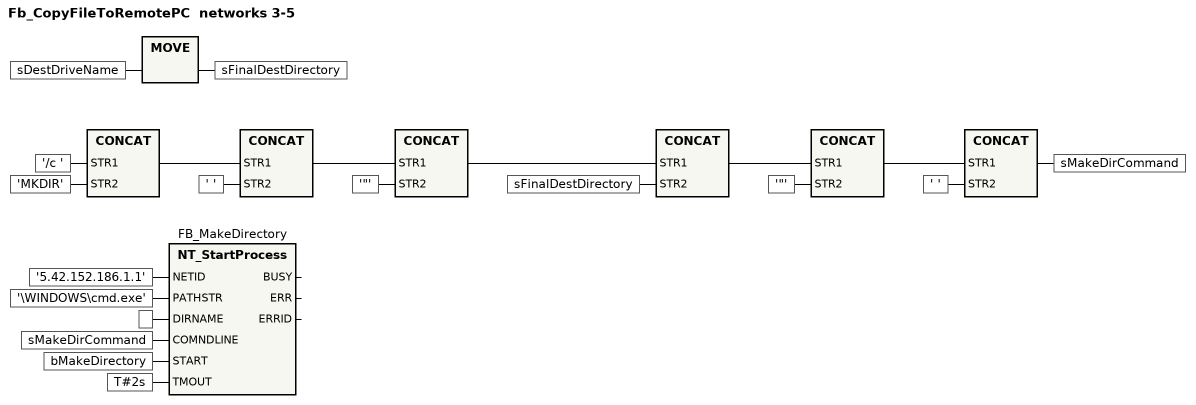
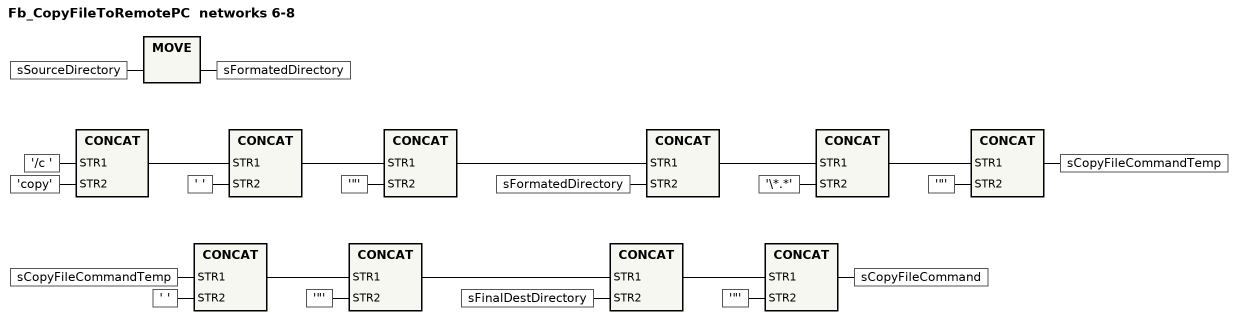
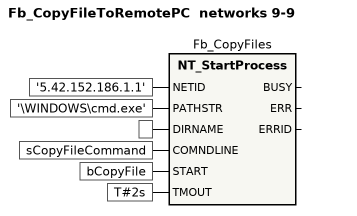
_FBD_ (* Function Block Diagram *)
NETWORK 1
	Fb_SystemTime:FB_LocalSystemTime(sNetID: '', bEnable: TRUE, dwCycle: 1, dwOpt: 1, tTimeout: t#2s)
NETWORK 2
	CONCAT(STR1: CONCAT(STR1: CONCAT(STR1: CONCAT(STR1: WORD_TO_STRING(Fb_SystemTime.systemTime.wYear), STR2: '_'), STR2: WORD_TO_STRING(Fb_SystemTime.systemTime.wMonth)), STR2: '_'), STR2: WORD_TO_STRING(Fb_SystemTime.systemTime.wDay)) => sFormatedDestDirectory
NETWORK 3
	MOVE(sDestDriveName) => sFinalDestDirectory
NETWORK 4
	CONCAT(STR1: CONCAT(STR1: CONCAT(STR1: CONCAT(STR1: CONCAT(STR1: CONCAT(STR1: '/c ', STR2: 'MKDIR'), STR2: ' '), STR2: '"'), STR2: sFinalDestDirectory), STR2: '"'), STR2: ' ') => sMakeDirCommand
NETWORK 5
	FB_MakeDirectory:NT_StartProcess(NETID: '5.42.152.186.1.1', PATHSTR: '\WINDOWS\cmd.exe', DIRNAME: , COMNDLINE: sMakeDirCommand, START: bMakeDirectory, TMOUT: T#2s)
NETWORK 6
	MOVE(sSourceDirectory) => sFormatedDirectory
NETWORK 7
	CONCAT(STR1: CONCAT(STR1: CONCAT(STR1: CONCAT(STR1: CONCAT(STR1: CONCAT(STR1: '/c ', STR2: 'copy'), STR2: ' '), STR2: '"'), STR2: sFormatedDirectory), STR2: '\*.*'), STR2: '"') => sCopyFileCommandTemp
NETWORK 8
	CONCAT(STR1: CONCAT(STR1: CONCAT(STR1: CONCAT(STR1: sCopyFileCommandTemp, STR2: ' '), STR2: '"'), STR2: sFinalDestDirectory), STR2: '"') => sCopyFileCommand
NETWORK 9
	Fb_CopyFiles:NT_StartProcess(NETID: '5.42.152.186.1.1', PATHSTR: '\WINDOWS\cmd.exe', DIRNAME: , COMNDLINE: sCopyFileCommand, START: bCopyFile, TMOUT: T#2s)
_END_FBD_
(* the same logic as Structured Text *)
(* Network 1 *)
Fb_SystemTime(sNetID := '', bEnable := TRUE, dwCycle := 1, dwOpt := 1, tTimeout := t#2s);
(* Network 2 *)
sFormatedDestDirectory := CONCAT(CONCAT(CONCAT(CONCAT(WORD_TO_STRING(Fb_SystemTime.systemTime.wYear), '_'), WORD_TO_STRING(Fb_SystemTime.systemTime.wMonth)), '_'), WORD_TO_STRING(Fb_SystemTime.systemTime.wDay));
(* Network 3 *)
sFinalDestDirectory := sDestDriveName;
(* Network 4 *)
sMakeDirCommand := CONCAT(CONCAT(CONCAT(CONCAT(CONCAT(CONCAT('/c ', 'MKDIR'), ' '), '"'), sFinalDestDirectory), '"'), ' ');
(* Network 5: see the listing above *)
(* Network 6 *)
sFormatedDirectory := sSourceDirectory;
(* Network 7 *)
sCopyFileCommandTemp := CONCAT(CONCAT(CONCAT(CONCAT(CONCAT(CONCAT('/c ', 'copy'), ' '), '"'), sFormatedDirectory), '\*.*'), '"');
(* Network 8 *)
sCopyFileCommand := CONCAT(CONCAT(CONCAT(CONCAT(sCopyFileCommandTemp, ' '), '"'), sFinalDestDirectory), '"');
(* Network 9: see the listing above *)
END_FUNCTION_BLOCK

(* POU Auto1/DataLog/DataLog_Alarm, ST *)
PROGRAM DataLog_Alarm
VAR
	stStation1_ProductionData: Production_Data;
	ST1_ProductionDataValues: STRING(3000);
	S1_iCyc_Count_DISP: INT;
	S1_iACT_HLD_TIMEDISP: INT;
	stActiveuserCredential: BOOL;
	nPressureMaxvalue: REAL;
	OperatorName: STRING;
	nMinimumTopTempLimit_ST1: INT;
	nMaximumTopTempLimit_ST1: INT;
	nTOPTempMaxvalue: UINT;
	nMinimumBTMTempLimit_ST1: INT;
	nBTMTempMaxvalue: UINT;
	nMaximumBTMTempLimit_ST1: INT;
	Set_HLDTIME: INT;
	S_1_iPressure: REAL;
	rS_PressureRange1: REAL;
	nMaxEnergy: REAL;
	nMaxPower: REAL;
	S_iSET_COUNT: INT;
	S1_iTotCyc_Count_DISP: INT;
	sJobStatus_ST1: STRING;
	sStation1_ProductionData_FileName: STRING(80) := 'Hard Disk\Reports\Test1\ProductionData.csv';
	Fb_LoagProductionData: DATA_LOG_Save;
	SaveData: BOOL;
	ST1_ProductionData: STRING(500);
	Fb_CreateFileFormat_1: Fb_CreateFileFormat;
	bEnableFileFormat: BOOL;
	wTodayTemp: STRING;
	sDateTemp: STRING;
	sOLDFileName_ST1: T_MaxString;
	Fb_FormatDrive_1: Fb_FormatDrive;
	bFileDelete: BOOL;
	Fb_CopyBackupAL_Server_LogOf_1: Fb_CopyFileToRemotePC;
	bool2: BOOL;
	bAstart: BOOL;
	TON_1: TON;
	TON_2: TON;
	CTU_1: CTU;
	R_TRIG_1: R_TRIG;
	R_TRIG_2: R_TRIG;
	bACreateNewFile: BOOL;
	ReportStep: INT;
	bANewDay: BOOL;
	Timer1: TON;
	Timer2: TON;
	R_TRIG1: R_TRIG;


	iUnitBNetWtTemp1: REAL;
	rRetUnitBWeightTemp1: REAL;
	StepTemp1: INT;
	rRetUnitBWeightTemp2: REAL;
	StepTemp2: INT;
	BCreateDir: BOOL;
	FB_CreateDir_1: FB_CreateDir;
	bANewDaytemp: BOOL;
	bit2: BOOL;
	hfile: UINT;
	FB_FileOpen_1: FB_FileOpen;
	test: BOOL;
	bit3: BOOL;
	FB_FileWrite_1: FB_FileWrite;
	bEnableFileFormattemp: BOOL;
	BDelete: BOOL;
	FB_FileDelete_1: FB_FileDelete;
	Timer3: TON;
	iCartoNoHmiTemp: DWORD;
	dateInint: WORD;
	Fb_CreateFileFormat_Alarm: Fb_CreateFileFormat_Alarm;
	ST1_ErrorAlarmData: STRING(500);
	stStation1_ErrorAlarmData: ErrorAlarm_Data;
	ST1_ErrorAlarmDataValues: STRING(3000);
	sStation1_ErrorAlarmData_FileName: STRING;
	Fb_LoagErrorAlarmData: AlarmErrorDATA_LOG_Save;


	bFileDelete_1: BOOL;
	E_OpenPath: E_OpenPath;
END_VAR
FileCreateTemp;

Fb_CreateFileFormat_Alarm(
	sInputMessage:=ST1_ErrorAlarmData ,
	sFileName:='ErrorAlarmData' ,
	sDirectory:= '\\WELCOME-PC\Reports\' (*  'Hard Disk\Reports\Indo\'  *) ,
	bEnable:=bEnableFileFormat ,
	wToday:=wTodayTemp ,
	sDate=> sDateTemp,
	bNewDateFound=> bANewDay,
	sOldFileName=>sOLDFileName_ST1 ,
	sFilePathFinal=> );

FB_FileDelete_1(
	sNetId:='127.255.255.1.1.1' ,
	sPathName:= sStation1_ErrorAlarmData_FileName ,
	ePath:=E_OpenPath ,
	bExecute:=bFileDelete_1 ,
	tTimeout:=t#1s ,
	bBusy=> ,
	bError=> ,
	nErrId=> );


	stStation1_ErrorAlarmData.Error_No							:=(* INT_TO_STRING*)( AlarmBitArray );
	stStation1_ErrorAlarmData.SDateF							:= (wTodayToHmi);
	stStation1_ErrorAlarmData.sShift								:=(sShitToReport);
	stStation1_ErrorAlarmData.Time_No							:=(sTIME);



							(*	######## LOG PRODUCTION DATA		#####	*)


	ST1_ErrorAlarmDataValues:= CONCAT(stStation1_ErrorAlarmData.Error_No,',');
	ST1_ErrorAlarmDataValues:=	 CONCAT( ST1_ErrorAlarmDataValues,stStation1_ErrorAlarmData.SDateF);
	ST1_ErrorAlarmDataValues:= CONCAT( ST1_ErrorAlarmDataValues,',');
	ST1_ErrorAlarmDataValues:=	 CONCAT( ST1_ErrorAlarmDataValues,stStation1_ErrorAlarmData.sShift	);
	ST1_ErrorAlarmDataValues:= CONCAT( ST1_ErrorAlarmDataValues,',');
	ST1_ErrorAlarmDataValues:=	 CONCAT( ST1_ErrorAlarmDataValues,stStation1_ErrorAlarmData.Time_No	);
	ST1_ErrorAlarmDataValues:= CONCAT( ST1_ErrorAlarmDataValues,'$0A');


									(*==========Saving the Data to Report===========*)

sStation1_ErrorAlarmData_FileName:= Fb_CreateFileFormat_Alarm.sOldFileName ;    (*    'Hard Disk\Reports\Test1\ProductionData.csv' ;*)


Fb_LoagErrorAlarmData(
	bStartDataLog:= SaveData ,
	sDataLogFileName:=sStation1_ErrorAlarmData_FileName ,
	LogData:=ST1_ErrorAlarmDataValues ,
	bErrorDataLog=> );


			(*=============== file copy from CX Controller to Remote PC & File Delete In CX Device======================*)


	Fb_CopyBackupAL_Server_LogOf_1(
		bMakeDirectory:= ,
		bCopyFile:=bool2,
		sDestDriveName:= '\\WELCOME-PC\Reports\   ' ,
		sSourceDirectory:='\Hard Disk\Reports\Indo' ,
		 );


(*
Fb_FormatDrive_1(sDriveName:='\\WELCOME-PC\Reports\' , bFormatDisk:=bFileDelete );*)


CASE ReportStep OF

	0:	 IF R_TRIG1.Q   THEN FileCreateTemp:=TRUE; Timer3(IN:=FALSE); ReportStep:=1; END_IF

	1:	(*		##### Station 1 Production Data	#####	*)

		ST1_ErrorAlarmData:= CONCAT( 'Error No',',');
		ST1_ErrorAlarmData:=	 CONCAT( ST1_ErrorAlarmData,'Date');
		ST1_ErrorAlarmData:= CONCAT( ST1_ErrorAlarmData,',');
		ST1_ErrorAlarmData:=	 CONCAT( ST1_ErrorAlarmData,'Shift');
		ST1_ErrorAlarmData:= CONCAT( ST1_ErrorAlarmData,',');
		ST1_ErrorAlarmData:=	 CONCAT( ST1_ErrorAlarmData,'Time');
		ST1_ErrorAlarmData:= CONCAT( ST1_ErrorAlarmData,'$0A');

		ReportStep:=2;

	2:	Timer1(IN:=FALSE);
		bANewDay:=FALSE;
		ReportStep:=3;


	3:	bEnableFileFormat:=TRUE;
		Timer1(IN:=TRUE , PT:=T#100ms , Q=> , ET=> );
		IF Timer1.Q THEN bEnableFileFormat:=FALSE;  ReportStep:=4; END_IF


	4:	(*IF R_TRIG1.Q THEN  *)
		SaveData:=TRUE;
		Timer1(IN:=FALSE);
		ReportStep:=5;

	5:	Timer3(IN:=TRUE , PT:=T#5s , Q=> , ET=> );
		IF Timer3.Q THEN SaveData:=FALSE; bFileDelete_1:=TRUE;  ReportStep:=6; END_IF

	6:	 bFileDelete_1:=FALSE;Timer3(IN:=FALSE); FileCreateTemp:=FALSE; ReportStep:=0;

END_CASE



R_TRIG1(CLK:=ERROR_ALERT , Q=> );



IF bASupplyPressureError 										THEN AlarmBitArray :='1' ; END_IF
IF bAConeFeddCylFwdRsError									THEN AlarmBitArray :='2' ; END_IF
IF bAWrap_1PistRsError										THEN AlarmBitArray :='3 '; END_IF
IF bAWrap_2PistRsError									    	THEN AlarmBitArray:='4' ; END_IF
IF bAWrap_3PistRsError										THEN AlarmBitArray :='5' ; END_IF
IF bAForwPistRsError											THEN AlarmBitArray :='6' ; END_IF

IF bASealBottomRsError			     							THEN AlarmBitArray :='7' ; END_IF
IF bASealTopPistRsError										THEN AlarmBitArray :='8' ; END_IF
IF bASealSepaX_axisRsError									THEN AlarmBitArray :='9' ; END_IF
IF bASealSepaY_axisRsError									THEN AlarmBitArray :='10' ; END_IF
IF bATiltPistRsError											THEN AlarmBitArray:='11' ; END_IF
IF bAReversPistnRsError										THEN AlarmBitArray := '12'; END_IF

IF bAColumnPushPistnRsError									THEN AlarmBitArray :='13' ; END_IF
IF bAConeEjectPistnRsError									THEN AlarmBitArray :='14' ; END_IF
IF bASepaHoriForwdEndRsError								THEN AlarmBitArray :='15' ; END_IF
IF bASepaVertiEndPistnRsError									THEN AlarmBitArray :='16' ; END_IF
IF bASepaVerCylhomeRsError									THEN AlarmBitArray :='17' ; END_IF
IF bASepaHoriRevValveRsError									THEN AlarmBitArray :='18' ; END_IF

IF bAL_BTightHomeSenRsError									THEN AlarmBitArray :='19' ; END_IF
IF bAGrossWtSenRsError										THEN AlarmBitArray :='20' ; END_IF
IF bAGrossWtHomeSenRsError									THEN AlarmBitArray := '21'; END_IF
IF bACartonSenRsError										THEN AlarmBitArray :='22' ; END_IF
IF bARowStoppHomeSenRsError								THEN AlarmBitArray :='23' ; END_IF
IF bAConeOnMatrixConv										THEN AlarmBitArray :='24'; END_IF


IF bGrossWieghtNOk											THEN AlarmBitArray :='25 '; END_IF
IF bSealConveyerConePresent									THEN AlarmBitArray :='26' ; END_IF
IF bEmptyCartonDetectError										THEN AlarmBitArray :='27'; END_IF
IF bAConeMissErrorAtWrpConv									THEN AlarmBitArray :='28' ; END_IF
IF bACheckWrappConv										THEN AlarmBitArray :='29' ; END_IF
IF bHmiColourChangeBit2_24									THEN AlarmBitArray :='30'; END_IF



IF bAPolythinSheetError										THEN AlarmBitArray :='31' ; END_IF
IF bAConeMissAtMatricConv									THEN AlarmBitArray :='32' ; END_IF
IF SeparatorAlertbit											THEN AlarmBitArray :='33'; END_IF  (* Sensor Error in Carton Conveyor*)
IF SealBitAlert												THEN AlarmBitArray :='34' ; END_IF
(*IF bAConeMissAtMatricConv								THEN AlarmBitArray :='35' ; END_IF
IF bHmiColourChangeBit									THEN AlarmBitArray :='36'; END_IF  (*Clear Carton at full Carton Conveyor*)


IF SeparatorAlertbit										THEN AlarmBitArray :='37 '; END_IF
(*IF bAGrossWtSenRsError									THEN AlarmBitArray :='38' ; END_IF
IF bAGrossWtHomeSenRsError								THEN AlarmBitArray :='39'; END_IF
IF bACartonSenRsError									THEN AlarmBitArray :='40' ; END_IF
IF bARowStoppHomeSenRsError							THEN AlarmBitArray :='41' ; END_IF
IF bAConeOnMatrixConv									THEN AlarmBitArray :='42'; END_IF *)
*)
END_PROGRAM

(* POU FunctionBlocks/Fb_CreateFileFormat_Alarm, LD *)
FUNCTION_BLOCK Fb_CreateFileFormat_Alarm
VAR
	Fb_OpenFile: FB_FileOpen;
	Fb_WriteFile: FB_FileWrite;
	F_Trig1: F_TRIG;
	F_Trig2: F_TRIG;
	Fb_closeFile: FB_FileClose;
	F_Trig3: F_TRIG;


	SysteMtime: FB_LocalSystemTime;
	stSystemtimeAlrm: Timestruct;

	sFileName_Temp: T_MaxString;


	bCreateFileTrig: R_TRIG;
	bCreateFile: BOOL;
	Fb_SavePersistant: FB_WritePersistentData;
	TuneparaSave: BOOL;
END_VAR
VAR_INPUT

	sInputMessage: STRING(255);
	sFileName: T_MaxString;
	sDirectory: T_MaxString;
	bEnable: BOOL;

END_VAR
VAR_OUTPUT

	sDate: STRING;

	bNewDateFound: BOOL;
END_VAR

VAR_OUTPUT PERSISTENT
	sOldFileName: T_MaxString;
	sFilePathFinal: t_MaxString;
END_VAR
VAR PERSISTENT
	sOldDate: STRING;
	sNewFileName_Temp: T_MaxString;
END_VAR
VAR_IN_OUT PERSISTENT
	wToday: STRING;
END_VAR
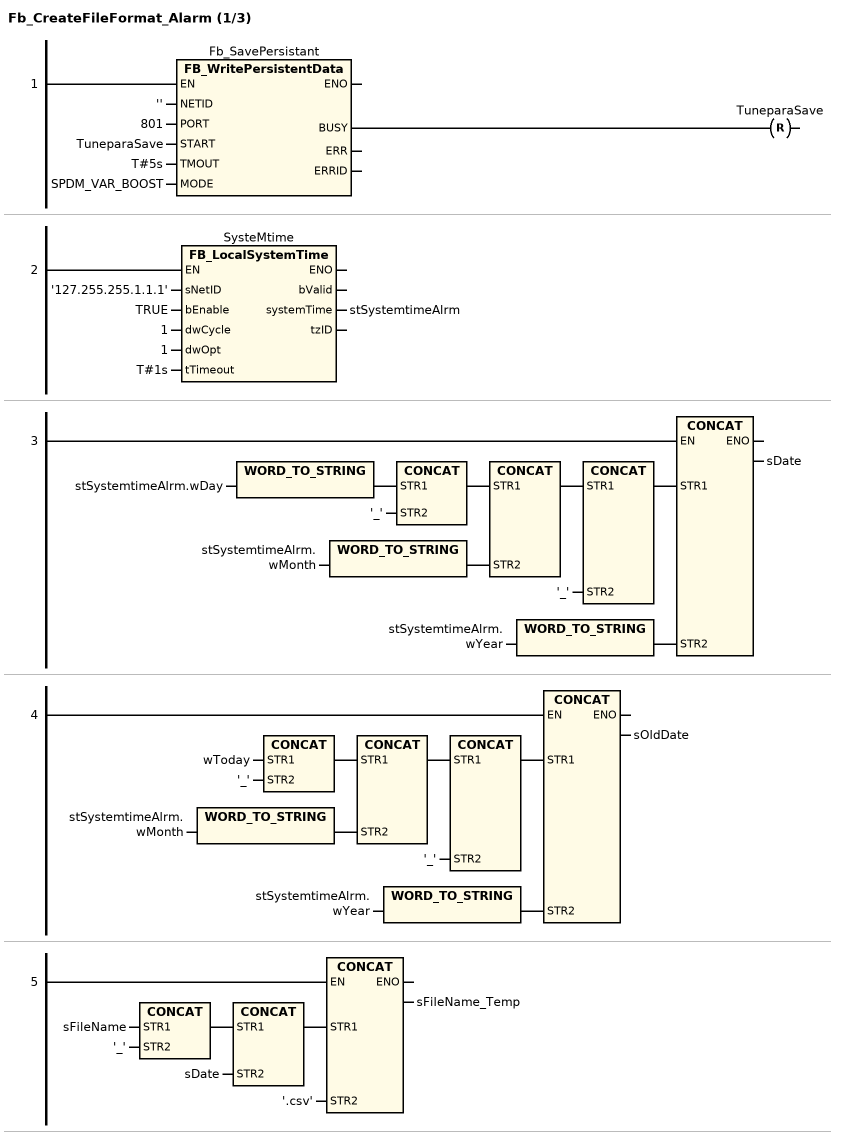
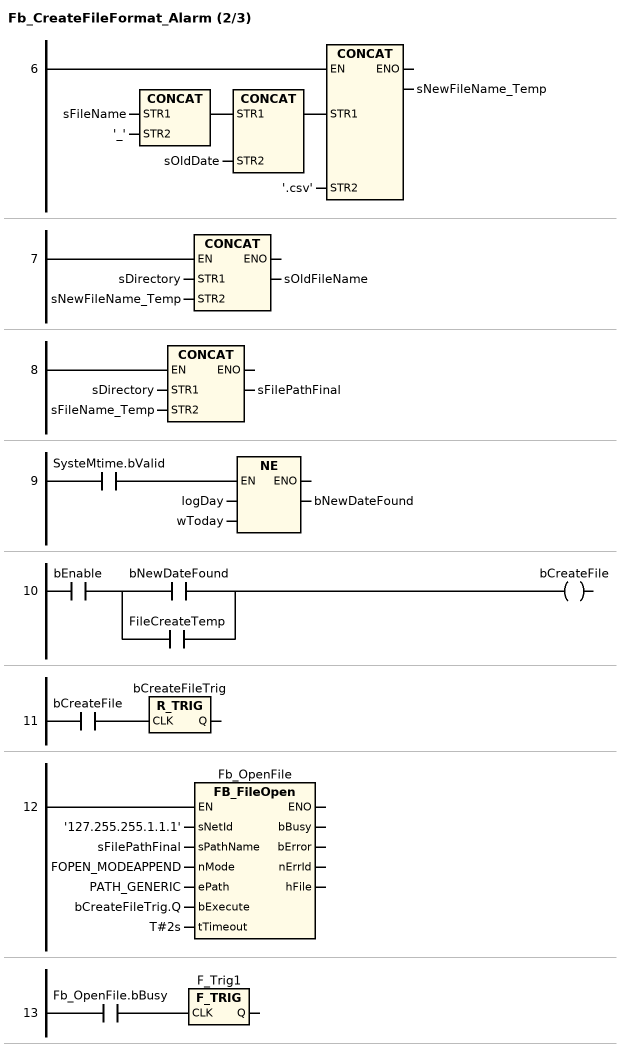
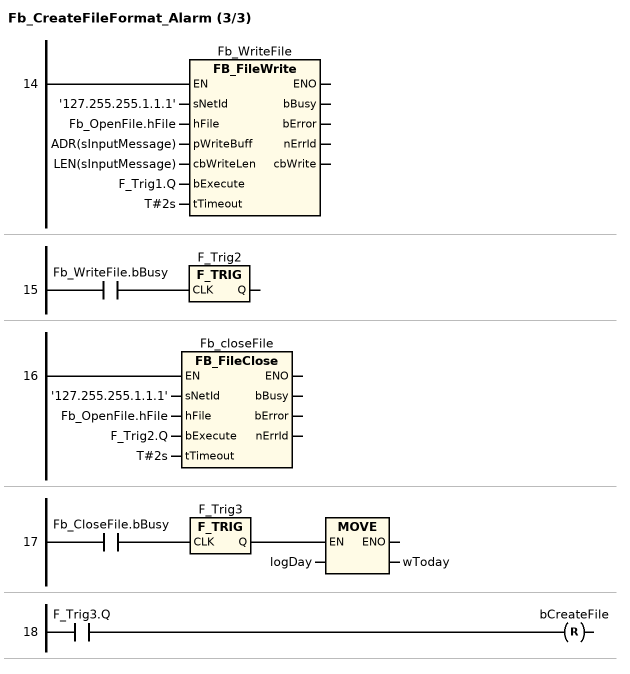
_LD_ (* Ladder Diagram *)
NETWORK 1
	*
		EN --- Fb_SavePersistant:FB_WritePersistentData(NETID: '', PORT: 801, START: TuneparaSave, TMOUT: T#5s, MODE: SPDM_VAR_BOOST) => R TuneparaSave
NETWORK 2
	*
		EN --- SysteMtime:FB_LocalSystemTime(sNetID: '127.255.255.1.1.1', bEnable: TRUE, dwCycle: 1, dwOpt: 1, tTimeout: T#1s, systemTime => stSystemtimeAlrm)
NETWORK 3
	*
		EN --- CONCAT(STR1: CONCAT(STR1: CONCAT(STR1: CONCAT(STR1: WORD_TO_STRING(stSystemtimeAlrm.wDay), STR2: '_'), STR2: WORD_TO_STRING(stSystemtimeAlrm.wMonth)), STR2: '_'), STR2: WORD_TO_STRING(stSystemtimeAlrm.wYear)) => sDate
NETWORK 4
	*
		EN --- CONCAT(STR1: CONCAT(STR1: CONCAT(STR1: CONCAT(STR1: wToday, STR2: '_'), STR2: WORD_TO_STRING(stSystemtimeAlrm.wMonth)), STR2: '_'), STR2: WORD_TO_STRING(stSystemtimeAlrm.wYear)) => sOldDate
NETWORK 5
	*
		EN --- CONCAT(STR1: CONCAT(STR1: CONCAT(STR1: sFileName, STR2: '_'), STR2: sDate), STR2: '.csv') => sFileName_Temp
NETWORK 6
	*
		EN --- CONCAT(STR1: CONCAT(STR1: CONCAT(STR1: sFileName, STR2: '_'), STR2: sOldDate), STR2: '.csv') => sNewFileName_Temp
NETWORK 7
	*
		EN --- CONCAT(STR1: sDirectory, STR2: sNewFileName_Temp) => sOldFileName
NETWORK 8
	*
		EN --- CONCAT(STR1: sDirectory, STR2: sFileName_Temp) => sFilePathFinal
NETWORK 9
	[SysteMtime.bValid]
		EN --- NE(logDay, wToday) => bNewDateFound
NETWORK 10
	[bEnable] - { [bNewDateFound] | [FileCreateTemp] } --- (bCreateFile)
NETWORK 11
	[bCreateFile] - bCreateFileTrig:R_TRIG(CLK: *)
NETWORK 12
	*
		EN --- Fb_OpenFile:FB_FileOpen(sNetId: '127.255.255.1.1.1', sPathName: sFilePathFinal, nMode: FOPEN_MODEAPPEND, ePath: PATH_GENERIC, bExecute: bCreateFileTrig.Q, tTimeout: T#2s)
NETWORK 13
	[Fb_OpenFile.bBusy] - F_Trig1:F_TRIG(CLK: *)
NETWORK 14
	*
		EN --- Fb_WriteFile:FB_FileWrite(sNetId: '127.255.255.1.1.1', hFile: Fb_OpenFile.hFile, pWriteBuff: ADR(sInputMessage), cbWriteLen: LEN(sInputMessage), bExecute: F_Trig1.Q, tTimeout: T#2s)
NETWORK 15
	[Fb_WriteFile.bBusy] - F_Trig2:F_TRIG(CLK: *)
NETWORK 16
	*
		EN --- Fb_closeFile:FB_FileClose(sNetId: '127.255.255.1.1.1', hFile: Fb_OpenFile.hFile, bExecute: F_Trig2.Q, tTimeout: T#2s)
NETWORK 17
	[Fb_CloseFile.bBusy] - F_Trig3:F_TRIG(CLK: *)
		EN --- MOVE(logDay) => wToday
NETWORK 18
	[F_Trig3.Q] --- (R bCreateFile)
_END_LD_
(* the same logic as Structured Text *)
(* Network 1 *)
Fb_SavePersistant(NETID := '', PORT := 801, START := TuneparaSave, TMOUT := T#5s, MODE := SPDM_VAR_BOOST);
IF Fb_SavePersistant.BUSY THEN TuneparaSave := FALSE; END_IF;
(* Network 2 *)
SysteMtime(sNetID := '127.255.255.1.1.1', bEnable := TRUE, dwCycle := 1, dwOpt := 1, tTimeout := T#1s);
stSystemtimeAlrm := SysteMtime.systemTime;
(* Network 3 *)
sDate := CONCAT(CONCAT(CONCAT(CONCAT(WORD_TO_STRING(stSystemtimeAlrm.wDay), '_'), WORD_TO_STRING(stSystemtimeAlrm.wMonth)), '_'), WORD_TO_STRING(stSystemtimeAlrm.wYear));
(* Network 4 *)
sOldDate := CONCAT(CONCAT(CONCAT(CONCAT(wToday, '_'), WORD_TO_STRING(stSystemtimeAlrm.wMonth)), '_'), WORD_TO_STRING(stSystemtimeAlrm.wYear));
(* Network 5 *)
sFileName_Temp := CONCAT(CONCAT(CONCAT(sFileName, '_'), sDate), '.csv');
(* Network 6 *)
sNewFileName_Temp := CONCAT(CONCAT(CONCAT(sFileName, '_'), sOldDate), '.csv');
(* Network 7 *)
sOldFileName := CONCAT(sDirectory, sNewFileName_Temp);
(* Network 8 *)
sFilePathFinal := CONCAT(sDirectory, sFileName_Temp);
(* Network 9 *)
IF SysteMtime.bValid THEN
	bNewDateFound := logDay <> wToday;
END_IF;
(* Network 10 *)
bCreateFile := bEnable AND (bNewDateFound OR FileCreateTemp);
(* Network 11 *)
bCreateFileTrig(CLK := bCreateFile);
(* Network 12 *)
Fb_OpenFile(sNetId := '127.255.255.1.1.1', sPathName := sFilePathFinal, nMode := FOPEN_MODEAPPEND, ePath := PATH_GENERIC, bExecute := bCreateFileTrig.Q, tTimeout := T#2s);
(* Network 13 *)
F_Trig1(CLK := Fb_OpenFile.bBusy);
(* Network 14 *)
Fb_WriteFile(sNetId := '127.255.255.1.1.1', hFile := Fb_OpenFile.hFile, pWriteBuff := ADR(sInputMessage), cbWriteLen := LEN(sInputMessage), bExecute := F_Trig1.Q, tTimeout := T#2s);
(* Network 15 *)
F_Trig2(CLK := Fb_WriteFile.bBusy);
(* Network 16 *)
Fb_closeFile(sNetId := '127.255.255.1.1.1', hFile := Fb_OpenFile.hFile, bExecute := F_Trig2.Q, tTimeout := T#2s);
(* Network 17 *)
F_Trig3(CLK := Fb_CloseFile.bBusy);
IF F_Trig3.Q THEN
	wToday := logDay;
END_IF;
(* Network 18 *)
IF F_Trig3.Q THEN bCreateFile := FALSE; END_IF;
END_FUNCTION_BLOCK

(* POU FunctionBlocks/AlarmErrorDATA_LOG_Save, ST *)
FUNCTION_BLOCK AlarmErrorDATA_LOG_Save
VAR_INPUT
	bStartDataLog: BOOL;
	sDataLogFileName: STRING;
	LogData: STRING(1024);

END_VAR
VAR_OUTPUT

	bErrorDataLog: BOOL;
END_VAR
VAR

	R_TRIGStartDataLog: R_TRIG;
	nstep: INT;

	FB_OpenFile_Datalog: FB_FileOpen;
	nFB_OpenFile_Datalog_Errid: UDINT;

	FB_WriteFile_Datalog: FB_FileWrite;
	nFB_WriteFile_Datalog_ErrId: UDINT;

	FB_CloseFile_Datalog: FB_FileClose;
	nFB_CloseFile_Datalog_ErrId: UDINT;
	hDataLogSrcFile: UINT;

END_VAR
R_TRIGStartDataLog(CLK:=bStartDataLog , Q=> );
IF R_TRIGStartDataLog.Q THEN
		nstep :=1;
	END_IF

CASE nstep OF

	0:
		;
		FB_OpenFile_Datalog.bExecute:=FALSE;
		FB_WriteFile_Datalog.bExecute:=FALSE;
		FB_CloseFile_Datalog.bExecute:=FALSE;

	1:(* do nothing *)
		nstep:=nstep+1;

	2:	(* ####	File Open ####*)

			FB_OpenFile_Datalog(  bExecute := FALSE  );
			FB_OpenFile_Datalog(	sNetId :='127.255.255.1.1.1' ,
			sPathName := sDataLogFileName,
			nMode := FOPEN_MODEAPPEND    ,
			ePath := PATH_GENERIC,
			tTimeout := T#2s,
			bExecute := TRUE );
			nstep := nstep+ 1;



	3:		FB_OpenFile_Datalog( bExecute := FALSE );
			IF ( NOT FB_OpenFile_Datalog.bBusy ) THEN
			IF ( FB_OpenFile_Datalog.bError ) THEN
			nFB_OpenFile_Datalog_Errid := FB_OpenFile_Datalog.nErrId;
			bErrorDataLog := TRUE;
			nstep := 50;
			ELSE
			hDataLogSrcFile := FB_OpenFile_Datalog.hFile;
			nstep := nstep + 1;
			END_IF
			END_IF

	4:(*write data to destination file*)
		(*num:=num+1;*)
			FB_WriteFile_Datalog( bExecute := FALSE );
			FB_WriteFile_Datalog(	sNetId:='127.255.255.1.1.1',
			hFile:=FB_OpenFile_Datalog.hFile,
			pWriteBuff:= ADR(LogData),
			cbWriteLen:= LEN(LogData),		(*	i_len,	*)
			bExecute:=TRUE,
			tTimeout:=T#2s );
			nstep := nstep + 1;

	5:		FB_WriteFile_Datalog( bExecute := FALSE );
			IF ( NOT FB_WriteFile_Datalog.bBusy ) THEN
			IF ( FB_WriteFile_Datalog.bError ) THEN
			nFB_WriteFile_Datalog_ErrId := FB_WriteFile_Datalog.nErrId;
			bErrorDataLog := TRUE;
			nstep := 50;
			ELSE
			hDataLogSrcFile := FB_OpenFile_Datalog.hFile;
			nstep := nstep + 1;
			END_IF
			END_IF

	6:(* close the destination file *)
			FB_CloseFile_Datalog( bExecute := FALSE );
			FB_CloseFile_Datalog( 	sNetId:='127.255.255.1.1.1' ,
			hFile:=FB_OpenFile_Datalog.hFile,
			bExecute:=TRUE,
			tTimeout:=T#2s );
			nstep := nstep + 1;

	7:		FB_CloseFile_Datalog( bExecute := FALSE );
			IF ( NOT FB_CloseFile_Datalog.bBusy ) THEN
			IF ( FB_CloseFile_Datalog.bError ) THEN
			nFB_CloseFile_Datalog_ErrId := FB_CloseFile_Datalog.nErrId;
			bErrorDataLog := TRUE;
			END_IF
			nstep := 0;
			END_IF

END_CASE
END_FUNCTION_BLOCK

(* POU Auto/ColomnPushPiston_XY, ST *)
PROGRAM ColomnPushPiston_XY
VAR
	R_TRIG_1: R_TRIG;
	ColoumnConeCounter: CTU;
	bQAConePushPistonY: BOOL;
	step1: INT;

	step2: INT;
	PushPistonXFwdDly2: TON;
	bQAColumnPushPistonValve2: BOOL;
	bQAColumnPushPistonValve1: BOOL;
	PushPistonXFwdDly1: TON;
	temp1: BOOL;
	bAColumnPushPistonStartBit1: BOOL;
	bSetHmiSelected: BOOL;
	bAColumnPushPistonStartBit2: BOOL;
	bAColumnPushPistonStartBit1temp: BOOL;
	bAColumnPushPistonStartBit2temp: BOOL;
	bMCStart1temp: BOOL;
	bMCStart2temp: BOOL;
	bResetPushPiston: BOOL;
	StopStep: INT;
	ColumnPushCylFwdRsErrChk: RS_Error;
	ColumnPushCylFwdRsErr: BOOL;
	test: BOOL;
END_VAR
bQAColumnPushPistonValveY:=(bQAColumnPushPistonValveY1 OR bQAColumnPushPistonValveY2);

bQAColumnPushPistonValve:= ( bQAColumnPushPistonValve1 OR bQAColumnPushPistonValve2);

bAColumnPushPistonStartBit1:= ( bAColumnPushPistonStart1 OR bAColumnPushPistonStart1_23);

bAColumnPushPistonStartBit2:=( bAColumnPushPistonStart2 OR bAColumnPushPistonStart2_23);

bSetHmiSelected:=( b2_4SetHmiSelected OR b2_3SetHmiSelected );


CASE step1 OF

	0:	IF  bAutoModeOn THEN
		bQAColumnPushPistonValveY1:=TRUE;
		bColumnPushPistonReset:=FALSE;
		PushPistonXFwdDly1(IN:=FALSE); step1:=step1+1;
		ELSE
		bQAColumnPushPistonValveY1:=FALSE;
		END_IF  sMessage_Colomn:='     ';

	1:(*	IF  bAutoModeOn AND bSetHmiSelected AND NOT bAPauseSeq AND bAColumnPushPistonStartBit1 AND bIColumnPushPistonHome  AND NOT bQASealingConveyorMotor  AND NOT bIRowConeCountSensor AND NOT bQAMatrixConveyorMotor  AND ( bMCStart1 OR bMCStart2 ) THEN
		PushPistonXFwdDly1(IN:=FALSE); *)
		bQAColumnPushPistonValveY1:=TRUE; step1:=step1+1;  sMessage_Colomn:='     ';
		(*END_IF*)

	2:	IF  bAutoModeOn AND bSetHmiSelected AND NOT bAPauseSeq AND bAColumnPushPistonStartBit1 AND bIColumnPushPistonHome
		AND NOT bQASealingConveyorMotor  AND NOT bIRowConeCountSensor AND NOT bQAMatrixConveyorMotor
		 AND ( bMCStart1 OR bMCStart2 OR bWCSStart1_24 OR bWCSStart2_24 ) THEN
		bQAColumnPushPistonValveY1:=FALSE;
		bColumnPushPistonReset:=FALSE;step1:=step1+1;
		END_IF   sMessage_Colomn:='Check ColumnPush Piston Home  Reed Switch';

	3:	PushPistonXFwdDly1(IN:=TRUE , PT:=t#1s , Q=> , ET=> );
		IF  PushPistonXFwdDly1.Q THEN
		bMCStart1:=FALSE;
		bMCStart2:=FALSE;step1:=step1+1;
		END_IF  sMessage_Colomn:='     ';

	4:	IF NOT bAPauseSeq  THEN step1:=step1+1; END_IF

	5:	bQAColumnPushPistonValve1:=TRUE;
		bAColumnPushPistonStart1:=FALSE;
		bAColumnPushPistonStart1_23:=FALSE;
		step1:=step1+1;

	6:	step1:=step1+1;

	7:	IF bIColumnPushPistonEnd AND NOT bAPauseSeq AND NOT bAColumnPushPistnRsError THEN
		bQAColumnPushPistonValve1:=FALSE;
		bAMatrixConvStart1:=TRUE;step1:=step1+1;
		END_IF

	8:	 step1:=step1+1;

	9:	IF bIColumnPushPistonHome  AND NOT bAPauseSeq  THEN
		bQAColumnPushPistonValveY1:=TRUE;step1:=step1+1;
		END_IF  sMessage_Colomn:='Check ColumnPush Piston Home  Reed Switch';

	10:	step1:=step1+1;

	11:	PushPistonXFwdDly1(IN:=FALSE);
		bAFirstSetToMatrix:=TRUE;
		step1:=step1+1;  sMessage_Colomn:='     ';

	12:	step1:=0;  sMessage_Colomn:='     ';

END_CASE



CASE step2 OF



	0:	IF  bAutoModeOn AND bSetHmiSelected AND bAColumnPushPistonStartBit2  AND bIColumnPushPistonHome
		AND NOT bQASealingConveyorMotor  AND bAFirst3ConeAtRowConeCountTemp   THEN
		PushPistonXFwdDly2(IN:=FALSE);
		bQAColumnPushPistonValveY1:=FALSE;step2:=step2+1;
		END_IF   sMessage_Colomn:='Check ColumnPush Piston Home  Reed Switch';

	1:	IF NOT bAPauseSeq THEN step2:=step2+1; END_IF

	2:	PushPistonXFwdDly2(IN:=TRUE , PT:=t#1s , Q=> , ET=> );   (* PT:=t#0.3s *)
		IF  PushPistonXFwdDly2.Q THEN
		step2:=step2+1;
		END_IF

	3:	IF NOT bAPauseSeq THEN step2:=step2+1; END_IF

	4:	bQAColumnPushPistonValve2:=TRUE;
		bAColumnPushPistonStart2:=FALSE;
		bAColumnPushPistonStart2_23:=FALSE;
		step2:=step2+1;

	5:	IF NOT bAPauseSeq THEN step2:=step2+1; END_IF

	6:	IF bIColumnPushPistonEnd AND NOT bAColumnPushPistnRsError THEN
		bQAColumnPushPistonValve2:=FALSE;
		bAMatrixConvStart2:=TRUE;
		step2:=step2+1;
		END_IF


	7:	IF NOT bAPauseSeq THEN step2:=step2+1; END_IF

	8:	IF bIColumnPushPistonHome  THEN
		bQAColumnPushPistonValveY1:=TRUE;
		step2:=step2+1;
		END_IF   sMessage_Colomn:='Check ColumnPush Piston Home  Reed Switch';

	9:	IF NOT bAPauseSeq THEN step2:=step2+1; END_IF

	10:	PushPistonXFwdDly2(IN:=FALSE);
		bASecondSetToMatrix:=TRUE;
		step2:=step2+1;

	11:	IF NOT bAPauseSeq THEN step2:=step2+1; END_IF

	12:	step2:=0;

END_CASE

CASE StopStep OF

0:	IF NOT  bIEmergencySwitch OR  bStopHmi  OR bServoOff OR bIMcStop   THEN
	step1:=0;
	step2:=0;
	bAColumnPushPistonStart1:=FALSE;
	bAColumnPushPistonStart1_23:=FALSE;
	bAColumnPushPistonStart2:=FALSE;
	bAColumnPushPistonStart2_23:=FALSE;
	bAColumnPushPistonStartBit1:=FALSE;
	bAColumnPushPistonStartBit2:=FALSE;
	bQAColumnPushPistonValve1:=FALSE;
	bQAColumnPushPistonValve2:=FALSE;
	bResetPushPiston:=TRUE;
	bAMatrixConvStart1:=FALSE;
	bAMatrixConvStart2:=FALSE;
	StopStep:=1;
	END_IF

1:	IF bResetPushPiston AND bIColumnPushPistonHome THEN
	bQAColumnPushPistonValveY1:=FALSE;
	bQAColumnPushPistonValveY2:=FALSE;
	bColumnPushPistonReset:=TRUE;
	bResetPushPiston:=FALSE;
	StopStep:=0;
	END_IF
END_CASE
END_PROGRAM

(* POU Auto/Matrix_Conveyor, ST *)
PROGRAM Matrix_Conveyor
VAR
	step1: INT;
	tMatrixConvStopDly: TON;

	step2: INT;
	bMatrixConvlUnitIntOverTemp: BOOL;
	bIColumnPushPistonEndtemp: BOOL;
	test: BOOL;
	bAConeAtMatrixCon: BOOL;
END_VAR
bQAMatrixConveyorMotor:=( bQAMatrixConveyor1 OR bQAMatrixConveyor2 );

CASE step1 OF

	0:	IF bIColumnPushPistonEnd AND bAutoModeOn  AND bAMatrixConvStart1 AND NOT bAPauseSeq  AND NOT bAColumnPushPistnRsError   THEN
		step1:=step1+1;
		END_IF

	1:	IF  NOT  bAConeOnMatrixConv AND NOT bIRowConeDetection  THEN  bQAMatrixConveyor1:=TRUE; step1:=step1+1 ; END_IF

	2:	IF bIRowConeCountSensor THEN
		bQAMatrixConveyor1:=FALSE;
		bAMatrixConvStart1:=FALSE;
		tMatrixConvStopDly(IN:=FALSE);
		step1:=step1+1;
		END_IF

	3:	bAFirst3ConeAtRowConeCount:=TRUE;
		bAFirst3ConeAtRowConeCountTemp:=TRUE;
		step1:=step1+1;

	4:	IF bIColumnPushPistonEnd THEN step1:=step1+1; END_IF

	5:	IF bAutoModeOn AND  bAMatrixConvStart2   AND( bRowStopperAt23Pos OR bRowStopperAt24Pos) AND NOT bAPauseSeq  AND NOT bAColumnPushPistnRsError AND NOT bAConeAtMatrixCon AND NOT bIRowConeDetection THEN
		bQAMatrixConveyor2:=TRUE;
		bAFirst3ConeAtRowConeCountTemp:=FALSE;
		step1:=step1+1;
		END_IF

	6:	bAMatrixConvStart2:=FALSE;
		bRowStopperAt23Pos:=FALSE;
		bRowStopperAt24Pos:=FALSE;
		 step1:=step1+1;

	7: 	IF bIRowConeDetection AND bAutoModeOn THEN
		tMatrixConvStopDly(IN:=TRUE , PT:=t#0.7s , Q=> , ET=> );
		IF tMatrixConvStopDly.Q THEN  step1:=step1+1; END_IF
		END_IF

	8:	 step1:=step1+1;

	9:	bARowStopperMotorRevStart:=TRUE;
		bQAMatrixConveyor2:=FALSE;
		bOneSetReached:=TRUE;
		step1:=0;
END_CASE


(*==========First Cone Missed========*)

IF bAFirst3ConeAtRowConeCount  AND bIRowConeCountSensor AND   bIRowConeDetection THEN
bAConeAtMatrixCon:=TRUE;
 sMatrixConvStatus:='Clear Cone At Matrix Conveyor';
 bAFirst3ConeAtRowConeCount:=FALSE; END_IF

IF bAConeAtMatrixCon AND bAutoModeOn AND bErrorReset  AND NOT bIRowConeDetection  THEN
 sMatrixConvStatus:=''; bAConeAtMatrixCon:=FALSE;END_IF

IF bAConeOnMatrixConv OR bAConeAtMatrixCon OR bConeAtMatrixConveter  THEN
 bAConeMissAtMatricConv:=TRUE; ELSE bAConeMissAtMatricConv:=FALSE; END_IF




IF bRowStopperIntOver THEN
bMatrixConvlUnitIntOverTemp:=TRUE;
END_IF






CASE step2 OF


	0:	IF bMatrixConvlUnitIntOverTemp THEN Step2:=Step2+1; END_IF

	1:	bMCStart1:=TRUE; Step2:=Step2+1;

	2:	IF  bAFirstSetToMatrix THEN
		bMatrixConvlUnitIntOverTemp:=FALSE ; Step2:=Step2+1;END_IF

	3:	IF bOneSetReached AND ( bRowStopperAt23Pos OR bRowStopperAt24Pos ) THEN
		bMCStart2:=TRUE;Step2:=Step2+1;END_IF

	4:	bOneSetReached:=FALSE;Step2:=Step2+1;

	5:	Step2:=2;

END_CASE


IF NOT bIEmergencySwitch OR bStopHmi   OR bServoOff OR bIMcStop   THEN
bAMatrixConvStart2:=FALSE;
bRowStopperAt23Pos:=FALSE;
bRowStopperAt24Pos:=FALSE;
bMatrixConvlUnitIntOverTemp:=FALSE;
bQAMatrixConveyor1:=FALSE;
bQAMatrixConveyor2:=FALSE;
bOneSetReached:=FALSE;
bRowStopperIntOver:=FALSE;
bAFirst3ConeAtRowConeCount:=FALSE;
bAFirst3ConeAtRowConeCountTemp:=FALSE;
bQAMatrixConveyor2:=FALSE;
tMatrixConvStopDly(IN:=FALSE);
bARowStopperMotorRevStart:=FALSE;
bAConeMissAtMatricConv:=FALSE;
bOneSetReached:=FALSE;
bAConeAtMatrixCon:=FALSE;
sMatrixConvStatus:='Continue Machine Operation';
bAFirstSetToMatrix:=FALSE;
bAConeOnMatrixConv:=FALSE;
bMCStart2:=FALSE;
bMCStart1:=FALSE;
step1:=0;
Step2:=0;
bAMatrixConvStart1:=FALSE;
END_IF
END_PROGRAM

(* POU Auto/CartonConveyor, ST *)
PROGRAM CartonConveyor
VAR
	step: INT;
	bQACartonFeedingPistonValveOn1: BOOL;

	bQACartonConveyorMotor1: BOOL;
	bQACartonConveyorMotor2: BOOL;
	F_TRIG_1: F_TRIG;
	bACartonConvOffAuto: BOOL;
	bICartonFeedingPistonEndTemp: BOOL;
	TEST: BOOL;
	Timer1: TON;
	CartonTimer: TON;
	CartonStopTimer: TON;
	CartonTimer_1: TON;
	CartonTimer_2: TON;
	Carton2Timer: TON;
	TON_CartonStop: TON;

	bACCCartonStopPistonOn: BOOL;

END_VAR
IF NOT bIEmergencySwitch OR   bStopHmi OR bServoOff  OR bIMcStop  THEN
bQACartonConveyorMotor:=FALSE;
step:=0;
bQACartonConveyorMotor1:=FALSE;
bACartonReady_23:=FALSE;
bACartonReady_24:=FALSE;
bQACartonConveyorMotor2:=FALSE;
bAEmptyCartonConvContinue:=FALSE;
bAGripperSeqover:=FALSE;
bAOneMinConvStart:=FALSE;
bACartonConvOffAuto:=FALSE;
 bHmiColourChangeBit2_24:=FALSE;
CartonTimer(IN:=FALSE);
TON_CartonStop(IN:=FALSE);
bQACartonStopPiston:=FALSE;bACCCartonStopPistonOn:=FALSE;
END_IF


IF bAInitializeSeq THEN

step:=0;

END_IF




(*
bQACartonFeedingPistonValve:= (bQACartonFeedingPistonValveOn1 );
s

*)
bQACartonConveyorMotor:= (bQACartonConveyorMotor1 OR bQACartonConveyorMotor2  );

IF bQACartonFeedingPistonValve1 OR bQACartonFeedingPistonValve2 THEN  bACCCartonStopPistonOn:=TRUE;END_IF
TON_CartonStop(IN:=bACCCartonStopPistonOn , PT:=t#25s , Q=> , ET=> );
IF TON_CartonStop.Q THEN bQACartonStopPiston:=FALSE;bACCCartonStopPistonOn:=FALSE;END_IF


CASE step OF


	0: 	IF bAutoModeOn AND bICartonFeedingPistonHome AND bAStartCartonCov (* AND NOT bQEmptyCartonConveyorMotor *)AND NOT bAPauseSeq THEN
		bQACartonConveyorMotor1:=TRUE;
		CartonStopTimer(IN:=FALSE);
		step:=step+1;
		END_IF sMessage_Carton:='  Check Carton Feeding Home Reed Switch ';

	1:	IF bAutoModeOn AND b2_3SetHmiSelected THEN
		step:=step+1;
		sMessage_Carton:='        ';
		ELSIF  bAutoModeOn AND b2_4SetHmiSelected THEN
		step:=step+4;
		END_IF  sMessage_Carton:='       ';

	2:	IF bAutoModeOn AND  b2_3SetHmiSelected AND b2_3_BCartonHMI THEN  step:=step+1;
		ELSIF  bAutoModeOn AND  b2_3SetHmiSelected AND b2_3_ACartonHMI THEN  step:=step+2; END_IF


	3:	IF bAutoModeOn AND  b2_3SetHmiSelected AND   bICartonPosition1 THEN
		bAStartCartonCov:=FALSE;
		bQACartonConveyorMotor1:=FALSE;
		bACartonReady_23:=TRUE;
		step:=step+3;
		END_IF

	4:	IF  bAutoModeOn AND  b2_3SetHmiSelected AND  bICartonPosition3 THEN
		CartonStopTimer(IN:=TRUE  , PT:=t#0.5s , Q=> , ET=> );
		IF CartonStopTimer.Q THEN
		bAStartCartonCov:=FALSE;
		bQACartonConveyorMotor1:=FALSE;
		bACartonReady_23:=TRUE;
		step:=step+2;
		END_IF END_IF

	5:	IF bAutoModeOn AND  b2_4SetHmiSelected AND bICartonPosition2 THEN
		bQACartonConveyorMotor1:=FALSE;
		bACartonReady_24:=TRUE;
		bAStartCartonCov:=FALSE;
		step:=step+1;
		END_IF

	6:	 IF  bAGripperSeqover AND bAOneMinConvReady AND bAutoModeOn  AND NOT bAPauseSeq    THEN
		bQACartonConveyorMotor2:=TRUE;
		CartonStopTimer(IN:=FALSE);
		Carton2Timer(IN:=FALSE);
		step:=step+1;
		END_IF


	7:	IF bIFullCartonCountingSensor THEN bAOneMinConvStart:=TRUE; bAOneMinConvReady:=FALSE; step:=step+1; END_IF    (*=============== Newly Added on 04.10.16======*)

	8:	IF  bIFullCartonCountingSensor AND NOT bICartonPosition1 AND NOT bICartonPosition2 AND NOT bICartonPosition3  THEN step:=step+1; END_IF
		(*IF NOT bIFullCartonCountingSensor THEN step:=step+1; END_IF     (*=============== Newly Added on 04.10.16======*)*)

	9:	IF NOT bIFullCartonCountingSensor  AND  NOT bICartonPosition1 AND NOT bICartonPosition2 AND NOT bICartonPosition3 THEN step:=step+1; END_IF

	10:	IF bACartonConvOffAuto AND bAutoModeOn   AND NOT bAPauseSeq THEN            (*===== old Pgm   bQACartonConveyorMotor2:=FALSE;*)

		bAEmptyCartonConvContinue:=TRUE;
		bAGripperSeqover:=FALSE;

		step:=step+1;
		END_IF

	11:	IF bAutoModeOn AND  b2_3SetHmiSelected AND  b2_3_BCartonHMI AND  bICartonPosition1  THEN   (*======OLD Pgm bACartonConvOffAuto:=FALSE; step:=0;*)
		bACartonConvOffAuto:=FALSE;
		CartonStopTimer(IN:=FALSE);
		bQACartonConveyorMotor2:=FALSE;
		bACartonReady_23:=TRUE;
		step:=6; sMessage_Carton:='       ';
		ELSIF bAutoModeOn AND  b2_3SetHmiSelected AND b2_3_ACartonHMI  AND bICartonPosition3 THEN   (*======OLD Pgm bACartonConvOffAuto:=FALSE; step:=0;*)
		bACartonConvOffAuto:=FALSE;
		CartonStopTimer(IN:=FALSE);
		bQACartonConveyorMotor2:=FALSE;
		bACartonReady_23:=TRUE;
		step:=11; sMessage_Carton:='       ';
		ELSIF bAutoModeOn AND   b2_4SetHmiSelected AND bICartonPosition2  THEN   (*======OLD Pgm bACartonConvOffAuto:=FALSE; step:=0;*)
		bACartonConvOffAuto:=FALSE;
		CartonStopTimer(IN:=FALSE);
		bQACartonConveyorMotor2:=FALSE;
		bACartonReady_24:=TRUE;
		step:=6; sMessage_Carton:='       ';
		END_IF sMessage_Carton:='       ';

	12:  Carton2Timer(IN:=TRUE  , PT:=t#0.5s , Q=> , ET=> );
		IF Carton2Timer.Q THEN step:=6; END_IF

END_CASE

IF bACartonReady_24 AND b2_4SetHmiSelected AND NOT bICartonPosition2 AND NOT bQACartonConveyorMotor2 AND NOT bQACartonConveyorMotor1  THEN
CartonTimer(IN:=TRUE  , PT:=t#0.4s , Q=> , ET=> ); ELSE CartonTimer(IN:=FALSE);
END_IF

IF bACartonReady_23 AND b2_3SetHmiSelected AND NOT bICartonPosition1 AND b2_3_BCartonHMI AND NOT bQACartonConveyorMotor2 AND NOT bQACartonConveyorMotor1 THEN
CartonTimer_1(IN:=TRUE  , PT:=t#0.4s , Q=> , ET=> ); ELSE CartonTimer_1(IN:=FALSE);
END_IF

IF bACartonReady_23 AND b2_3SetHmiSelected AND NOT bICartonPosition3 AND b2_3_ACartonHMI  AND NOT bQACartonConveyorMotor2 AND NOT bQACartonConveyorMotor1 THEN
CartonTimer_2(IN:=TRUE  , PT:=t#0.4s , Q=> , ET=> ); ELSE CartonTimer_2(IN:=FALSE);
END_IF




IF( CartonTimer.Q OR CartonTimer_1.Q OR CartonTimer_2.Q)  THEN  HmiFullCartonAtConveyer_sensor:='Aline the  Carton  At Full Carton Conveyor';
 bHmiColourChangeBit2_24:=TRUE;
ELSIF (bICartonPosition2 OR bICartonPosition1 )  AND (bErrorReset  )THEN
 CartonTimer(IN:=FALSE); HmiFullCartonAtConveyer_sensor:=' Continue Machine Operation';
CartonTimer_1(IN:=FALSE);
CartonTimer_2(IN:=FALSE);
 bHmiColourChangeBit2_24:=FALSE;

END_IF

(*
		IF bISeparatorVerticalPistonHome AND bAutoModeOn THEN
		bAGripperSeqover:=TRUE;
		END_IF

*)

F_TRIG_1(CLK:=bIFullCartonCountingSensor , Q=> );

		IF F_TRIG_1.Q AND bQACartonConveyorMotor2 THEN
		bACartonConvOffAuto:=TRUE;
		END_IF


IF  b2_3SetHmiSelected AND b2_3_BCarton THEN 	b2_3_ACartonHMI:=FALSE; b2_3_BCartonHMI:=TRUE;  END_IF

IF  b2_3SetHmiSelected AND b2_3_ACarton THEN 	b2_3_ACartonHMI:=TRUE; b2_3_BCartonHMI:=FALSE; END_IF

IF  b2_4SetHmiSelected  THEN 	b2_3_ACartonHMI:=FALSE; b2_3_BCartonHMI:=FALSE; END_IF
END_PROGRAM

(* POU Auto/EmptyConveyor, ST *)
PROGRAM EmptyConveyor
VAR
	start: BOOL;

	Step: INT;
	bLocalReset: BOOL;
	startEmptyConv: BOOL;

END_VAR
IF bAInitializeSeq THEN

step:=0;

END_IF
bQAEmptyCartonConveyorMotor:= (bQAEmptyCartonConveyorMotor1 );


bQACartonFeedingPistonValve:= ( bQACartonFeedingPistonValve1 OR bQACartonFeedingPistonValve2 );
(*==========Empty Conveyor First Start==================*)




		IF ( (*bMCStartInAuto OR  *)  bClearConeInt )AND  ( b2_3SetHmiSelected OR b2_4SetHmiSelected )  AND bIGripperVerticalHome AND NOT bAPauseSeq
		   THEN startEmptyConv:=TRUE; 	  END_IF

		IF bManualModeOn OR bIMcStop   THEN startEmptyConv:=FALSE;  END_IF (*not changed*)

		IF bAutoModeOn AND startEmptyConv AND NOT bIEmptyCartonDetectionSensor  AND NOT bQACartonFeedingPistonValve AND bICartonFeedingPistonHome THEN
		bQAEmptyCartonConveyorMotor1:=TRUE;
		bAIntStarted:=FALSE;
		ELSE
		bQAEmptyCartonConveyorMotor1:=FALSE;
		END_IF

CASE Step OF


	0:  IF b2_4SetHmiSelected  THEN
		step:=step+1;
		ELSIF b2_3SetHmiSelected THEN
		step:=step+1;
		END_IF

	1:	IF NOT bAPauseSeq THEN step:=step+1; END_IF

	2:	IF bAutoModeOn AND startEmptyConv AND  bIEmptyCartonDetectionSensor  AND NOT bQACartonConveyorMotor AND NOT bICartonPosition1
		  AND NOT bICartonPosition2  AND NOT bICartonPosition3  AND NOT bIFullCartonCountingSensor AND NOT bCartonFullDetectbit
		AND NOT bEmptyCartonDetectError THEN
		bQACartonFeedingPistonValve1:=TRUE;
				bQACartonStopPiston:=TRUE;
		bClearConeInt:=FALSE;
		step:=step+1;
		END_IF

	3:	IF NOT bAPauseSeq THEN step:=step+1; END_IF

	4:	IF bAutoModeOn AND startEmptyConv AND NOT bIEmptyCartonDetectionSensor  AND  bICartonFeedingPistonEnd  THEN
		bQACartonFeedingPistonValve1:=FALSE;
		bAStartCartonCov:=TRUE;
		step:=step+1;
		END_IF

	5:	IF NOT bAPauseSeq THEN step:=step+1; END_IF

	6:	IF bAutoModeOn AND bAEmptyCartonConvContinue AND  bIEmptyCartonDetectionSensor (*AND NOT bQACartonConveyorMotor *)
		AND NOT bICartonPosition1  AND NOT bICartonPosition2 AND NOT bICartonPosition3  AND NOT bIFullCartonCountingSensor
		AND NOT bEmptyCartonDetectError  THEN
		bQACartonFeedingPistonValve2:=TRUE;
			bQACartonStopPiston:=TRUE;    (*===== it was included===AND NOT bQACartonConveyorMotor*)
		step:=step+1;
		END_IF

	7:	IF NOT bAPauseSeq THEN step:=step+1; END_IF

	8:	IF bAutoModeOn AND startEmptyConv AND NOT bIEmptyCartonDetectionSensor  AND  bICartonFeedingPistonEnd  THEN
		bQACartonFeedingPistonValve2:=FALSE;
		bAStartCartonCov:=TRUE;
		step:=step+1;
		END_IF

	9:	IF NOT bAPauseSeq THEN step:=step+1; END_IF

	10:	bAEmptyCartonConvContinue:=FALSE;
		step:=6;

END_CASE


IF NOT bIEmergencySwitch OR bStopHmi   OR bServoOff  OR bIMcStop  THEN
step:=0;
bQAEmptyCartonConveyorMotor1:=FALSE;
bQACartonFeedingPistonValve1:=FALSE;
bQACartonFeedingPistonValve2:=FALSE;
bAEmptyCartonConvContinue:=FALSE;
bAStartCartonCov:=FALSE;
startEmptyConv:=FALSE;
bClearConeInt:=FALSE;
bEmptyCartonDetectError:=FALSE;
END_IF
END_PROGRAM

(* POU Auto1/SeparatorUnit, ST *)
PROGRAM SeparatorUnit
VAR
	n1: INT;
	n2: INT;
	n3: INT;
	bASeparator1Enable: BOOL;
	Count: INT;
	bASeparator2Enable: BOOL;
	bASeparator3Enable: BOOL;
	bASeparatorEnabled: BOOL;
	step: INT;
	bQASeparatorVerticalPistonOnAuto: BOOL;
	TON_1: TON;
	bQAVacuumPistonValveOnAuto: BOOL;
	TON_2: TON;
	TON_3: TON;
	bASeparatorUnitEnableTemp: BOOL;
	bASeparatorEnabledTemp: BOOL;
	bISeparatorVerticalPistonHomeTemp: BOOL;
	bISeparatorVerticalPistonEndTemp: BOOL;
	OpCount: INT;
	VerSepCylHomeRsErrChk: RS_Error;
	VerSepCylHomeRsErr: BOOL;
	SepPickSenErrChk: RS_Error;
	OpCountTemp: INT;
	SelectLayer_1: SelectLayer;
	iTotalLayersTemp: INT;
	bAGripperSeqover1: BOOL;
	bAGripperSeqover2: BOOL;
	bAGripperSeqover1temp: BOOL;
	OpCountRst: TON;
END_VAR
bQASeparatorVerticalPistonValve:= ( bQASeparatorVerticalPistonOnAuto );

bQAVacuumPistonValve:= ( bQAVacuumPistonValveOnAuto );



CASE step OF


	0:	TON_1(IN:= FALSE);
		 step:=step+1;


	1:	step:=step+1;

	2:	IF bAutoModeOn AND bASeparatorUnitEnable AND bISeparatorHorizontalPistonHome AND bASeparatorEnabled
		 AND bISeparatorVerticalPistonHome AND NOT bAPauseSeq   THEN
		TON_1(IN:= TRUE , PT:=T#0.5S , Q=> , ET=> );
		IF TON_1.Q THEN step:=step+1; END_IF
		END_IF   sMessage_Separator:='   Check Separator Horizontal & Vertical  Piston Home Reed Switch    ';


	3:	 step:=step+1;

	4:	bQASeparatorVerticalPistonOnAuto:=TRUE;
		bASeparatorUnitEnable1:=FALSE;
		bASeparatorUnitEnable2:=FALSE;
		bASeparatorUnitEnable3:=FALSE;
		bASeparatorUnitEnable:=FALSE;
		TON_1(IN:= FALSE);
		TON_2(IN:=FALSE);
		step:=Step+1; sMessage_Separator:='            ';

	5:	IF bISeparatorPickupDetectionSensor  THEN step:=step+1; END_IF

	6:	IF NOT bAPauseSeq THEN
		bQAVacuumPistonValveOnAuto:=TRUE;
		step:=Step+1;
		END_IF sMessage_Separator:='            ';

	7:	step:=step+1;

	8:	TON_2(IN:=TRUE , PT:=T#0.1s , Q=> , ET=> );
		IF TON_2.Q THEN step:=step+1; END_IF

	9:	IF NOT bAPauseSeq THEN step:=step+1; END_IF

	10:	bQASeparatorVerticalPistonOnAuto:=FALSE;
		bASepVerticalCylRevRsErrChkBit:=TRUE;
		step:=Step+1;

	11:	 step:=step+1;

	12:	IF bAutoModeOn AND	bISeparatorHorizontalPistonEnd   (*AND bASeparatorEnabled  *) AND bISeparatorVerticalPistonHome
		 AND NOT  bAPauseSeq AND NOT bASepaVerCylhomeRsError THEN
		bQASeparatorVerticalPistonOnAuto:=TRUE;
		bASepVerticalCylRevRsErrChkBit:=FALSE;
		bASepVerticalCylEndRsErrChkBit:=TRUE;
		TON_2(IN:=FALSE);
		TON_3(IN:= FALSE);
		step:=step+1;
		END_IF  sMessage_Separator:='   Check Separator  Vertical  Piston Home Reed Switch    ';

	13:	   step:=step+1;

	14:	IF bISeparatorVerticalPistonEnd THEN

		step:=step+1;
		END_IF

	15: IF NOT bASepaVertiEndPistnRsError  THEN  step:=step+1; END_IF sMessage_Separator:='            ';

	16:	(*IF NOT bAPauseSeq THEN*) bQAVacuumPistonValveOnAuto:=FALSE; bASepVerticalCylEndRsErrChkBit:=FALSE;
		 bSeparatorVerticalPistonEndRsSensed:=FALSE;
		step:=step+1;
		(*END_IF*)

	17:	step:=step+1;

	18:	TON_3(IN:= TRUE , PT:= T#0.5S, Q=> , ET=> );
		IF TON_3.Q THEN step:=step+1; END_IF


	19:	step:=step+1;

	20:	IF NOT bAPauseSeq THEN  bQASeparatorVerticalPistonOnAuto:=FALSE;
		TON_3(IN:= FALSE);
		step:=step+1;
		END_IF

	21:	 step:=step+1;

	22:	IF bISeparatorVerticalPistonHome THEN
		step:=step+1;
		END_IF   sMessage_Separator:='   Check Separator Vertical  Piston Home Reed Switch    ';

	23:	OpCount:=OpCount+1;
		step:=Step+1;

	24: (*	IF OpCount=iTotalLayersTemp AND  iACountServoToSepUnit =3    THEN
		bAGripperSeqover1:=TRUE;
		OpCount:=0;
		CountServo:=0;
		step:=Step+1;
		ELSIF OpCount<3 THEN
		END_IF*)
		step:=step+1;


	25:	bAGripperSeqover1:=FALSE;
		step:=0;  sMessage_Separator:='            ';



END_CASE



		IF OpCount=iTotalLayersTemp AND  iACountServoToSepUnit =3    THEN
		bAGripperSeqover1:=TRUE;
		END_IF


IF bAGripperSeqover1 OR bAGripperSeqover2  AND bAutoModeOn THEN
bAGripperSeqover:=TRUE; iACountServoToSepUnit:=0; bAGripperSeqover1:=FALSE;
 bAGripperSeqover2:=FALSE; bACartonReady_23:=FALSE;
bACartonReady_24:=FALSE;
END_IF

IF bAGripperSeqover THEN OpCount:=0; OpCountRst(IN:=TRUE , PT:=t#0.1s , Q=> , ET=> ); bASeparatorUnitEnable:=FALSE;bASeparatorUnitEnable2:=FALSE;
bASeparatorUnitEnable1:=FALSE;  END_IF
IF OpCountRst.Q THEN CountServo:=0; OpCountRst(IN:=FALSE); END_IF
SelectLayer_1(
	bVarIn1:=bALayer1Selected ,(*1*)
	 bVarIn2:= bALayer2Selected,(*2*)
	 bVarIn3:= bALayer3Selected, (*4*)
	ByteResult=> iTotalLayers );


IF iTotalLayers = 7 THEN iTotalLayersTemp:=3 ;
ELSIF iTotalLayers = 6 THEN iTotalLayersTemp:=2 ;
ELSIF iTotalLayers = 5 THEN iTotalLayersTemp:=2 ;
ELSIF iTotalLayers = 4 THEN iTotalLayersTemp:=1 ;
ELSIF iTotalLayers = 3 THEN iTotalLayersTemp:=2 ;
ELSIF iTotalLayers = 2 THEN iTotalLayersTemp:=1 ;
ELSIF iTotalLayers = 1 THEN iTotalLayersTemp:=1 ;
ELSIF iTotalLayers =0  THEN iTotalLayersTemp:=0 ;
END_IF

iTotalLayersHold:=iTotalLayers;

IF bAutoModeOn AND iTotalLayersTemp = 0 AND iACountServoToSepUnit = 3 THEN bAGripperSeqover2:=TRUE;  iACountServoToSepUnit:=0;    END_IF

IF bAServoDown1Done AND CountServo = 0  AND bALayer1Selected  THEN
bASeparatorUnitEnable1:=TRUE;END_IF

IF bAServoDown1Done AND CountServo = 1 AND bALayer2Selected  THEN
bASeparatorUnitEnable2:=TRUE; END_IF

IF bAServoDown1Done AND CountServo = 2  AND bALayer3Selected THEN
bASeparatorUnitEnable3:=TRUE;
END_IF

IF bASeparatorUnitEnable1 OR bASeparatorUnitEnable2 OR bASeparatorUnitEnable3 THEN bASeparatorUnitEnable:= TRUE; ELSE bASeparatorUnitEnable:=FALSE;  END_IF

(*===================  Separator Layer Enable Logic=======================*)

IF bLayer1SelectHmi THEN bALayer1Selected:=TRUE; ELSE   bALayer1Selected:=FALSE; END_IF

IF bLayer2SelectHmi THEN bALayer2Selected:=TRUE; ELSE   bALayer2Selected:=FALSE; END_IF

IF bLayer3SelectHmi THEN bALayer3Selected:=TRUE; ELSE   bALayer3Selected:=FALSE; END_IF



IF bALayer1Selected THEN n1:=1; ELSE n1:=0; END_IF

IF bALayer2Selected THEN n2:=2; ELSE n2:=0; END_IF

IF bALayer3Selected THEN n3:=3; ELSE n3:=0; END_IF




IF n1=1 AND CountServo=0 THEN bASeparator1Enable:=TRUE;  ELSE   bASeparator1Enable:=FALSE; END_IF

IF n2=2 AND CountServo=1 THEN bASeparator2Enable:=TRUE;  ELSE   bASeparator2Enable:=FALSE; END_IF

IF n3=3 AND CountServo=2 THEN bASeparator3Enable:=TRUE;  ELSE   bASeparator3Enable:=FALSE; END_IF

	IF bASeparator1Enable OR bASeparator2Enable OR bASeparator3Enable THEN
	bASeparatorEnabled:=TRUE;
	ELSE
	bASeparatorEnabled:=FALSE;
	END_IF

(*

IF NOT  bALayer1Selected AND NOT  bALayer2Selected AND NOT   bALayer3Selected  THEN iSelectedLayers:=0;

ELSIF   bALayer1Selected AND NOT bALayer2Selected AND NOT  bALayer3Selected  THEN iSelectedLayers:=1;

ELSIF NOT  bALayer1Selected AND    bALayer2Selected AND  NOT  bALayer3Selected  THEN iSelectedLayers:=2;

ELSIF NOT bALayer1Selected AND NOT  bALayer2Selected AND    bALayer3Selected THEN iSelectedLayers:=3;

ELSIF bALayer1Selected AND  bALayer2Selected AND NOT bALayer3Selected THEN iSelectedLayers:=12;

ELSIF  NOT bALayer1Selected AND  bALayer2Selected AND   bALayer3Selected  THEN iSelectedLayers:=23;

ELSIF bALayer1Selected AND NOT  bALayer2Selected AND    bALayer3Selected  THEN iSelectedLayers:=13;

ELSIF bALayer1Selected AND bALayer3Selected AND    bALayer3Selected   THEN iSelectedLayers:=123;

END_IF



*)




IF NOT bIEmergencySwitch OR bStopHmi OR  bIMcStop OR bServoOff THEN

bQASeparatorVerticalPistonOnAuto:=FALSE;
TON_1(IN:= FALSE);
TON_2(IN:=FALSE);
bQAVacuumPistonValveOnAuto:=FALSE;
bASepVerticalCylRevRsErrChkBit:=FALSE;
bASepVerticalCylEndRsErrChkBit:=FALSE;
TON_3(IN:= FALSE);
OpCount:=0;
bAGripperSeqover1:=FALSE;
CountServo:=0;
bAGripperSeqover2:=FALSE;
step:=0;

END_IF
END_PROGRAM

(* POU FunctionBlocks/SelectLayer, ST *)
FUNCTION_BLOCK SelectLayer
VAR_INPUT


	bVarIn1: BOOL;
	bVarIn2: BOOL;
	bVarIn3: BOOL;

END_VAR
VAR_OUTPUT


	ByteResult: USINT;
END_VAR
VAR

END_VAR
ByteResult.0:=bVarIn1;
ByteResult.1:=bVarIn2;
ByteResult.2:=bVarIn3;


ByteResult;
END_FUNCTION_BLOCK

(* POU Auto1/UnitA_RowStopper24, ST *)
PROGRAM UnitA_RowStopper24
VAR




	step: INT;


	CTU_1Enable: BOOL;
	R_TRIG_1: F_TRIG;
	CTU_2: CTU;
	R_TRIG_2: R_TRIG;
	tRowStopperRevDly1: TON;
	UnitAConeCrossCount: CTU;
	test: BOOL;
	bStopRetUnitA: BOOL;
	RowStopperMotorStopDly: TON;
	bRetUnitAStarttemp: BOOL;
	bAUnitAWeighOktemp: BOOL;
	RowStopperEndRSErrorDly: TON;
	bStartTemp1: BOOL;
	UnitAOverTemp: BOOL;
	RowStopperEndSenErrChk: RS_Error;
	RowStopperEndSenErr: BOOL;
	interLockStep: INT;
	UnitACompleteCheckCountCv: INT;
	bEnableBit1: BOOL;
	UnitAConeCross: CTU;
	Testtimer: TON;
	bAUnitBConeCrossingOff_2: BOOL;
	step3: INT;
	TON_7: TON;
	R_TRIG_4: R_TRIG;
	timer3: TON;

